KUKA KRL program: MyProgram_006().src

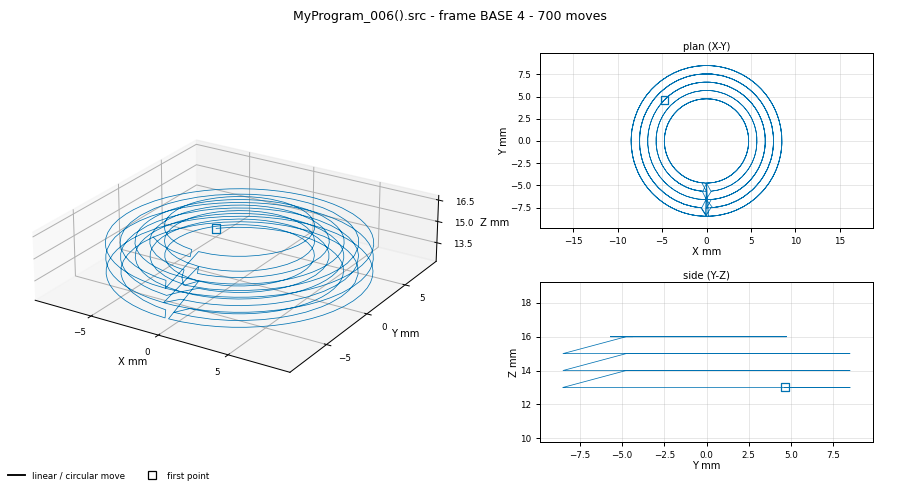
[picture p0: tool path of MyProgram_006().src in frame BASE 4, 700 of 700 moves have a stored position in this frame; points joined in program order, loops and branches not executed]
&ACCESS RVP
&REL 1
&PARAM TEMPLATE = C:\KRC\Roboter\Template\vorgabe
&PARAM EDITMASK = *
DEF MyProgram_006()
; ---- Setting reference (Base) ----
$BASE = BASE_DATA[4]

; --------------------------
; ---- Setting tool (TCP) ----
$TOOL = TOOL_DATA[3]
; --------------------------

$VEL.CP = VEL_APROX_PRINT
Startdeposition()
$VEL.CP = VEL_PRINT
LIN {X -4.726,Y 4.6339,Z 13,A -2.7634,B 0,C 0,E1 0.1598,E2 90.0717} C_DIS
LIN {X -4.1988,Y 5.116,Z 13,A -2.7237,B 0,C 0,E1 0.1598,E2 90.0718} C_DIS
LIN {X -3.6242,Y 5.5404,Z 13,A -2.6847,B 0,C 0,E1 0.1598,E2 90.0719} C_DIS
LIN {X -3.0059,Y 5.8983,Z 13,A -2.6468,B 0,C 0,E1 0.1598,E2 90.0719} C_DIS
LIN {X -2.0359,Y 6.3027,Z 13,A -2.5939,B 0,C 0,E1 0.1598,E2 90.072} C_DIS
LIN {X -1.1961,Y 6.5108,Z 13,A -2.5542,B 0,C 0,E1 0.1598,E2 90.0721} C_DIS
LIN {X -0.51,Y 6.6014,Z 13,A -2.5251,B 0,C 0,E1 0.1598,E2 90.0722} C_DIS
LIN {X 0.1819,Y 6.6196,Z 13,A -2.4988,B 0,C 0,E1 0.1598,E2 90.0722} C_DIS
LIN {X 0.8718,Y 6.5629,Z 13,A -2.4757,B 0,C 0,E1 0.1598,E2 90.0722} C_DIS
LIN {X 1.5516,Y 6.4333,Z 13,A -2.4561,B 0,C 0,E1 0.1598,E2 90.0722} C_DIS
LIN {X 2.2156,Y 6.238,Z 13,A -2.4398,B 0,C 0,E1 0.1598,E2 90.0722} C_DIS
LIN {X 2.8549,Y 5.9732,Z 13,A -2.4274,B 0,C 0,E1 0.1598,E2 90.0722} C_DIS
LIN {X 3.4624,Y 5.6414,Z 13,A -2.419,B 0,C 0,E1 0.1598,E2 90.0722} C_DIS
LIN {X 4.032,Y 5.2483,Z 13,A -2.4146,B 0,C 0,E1 0.1598,E2 90.0722} C_DIS
LIN {X 4.5579,Y 4.7985,Z 13,A -2.4143,B 0,C 0,E1 0.1598,E2 90.0722} C_DIS
LIN {X 5.0373,Y 4.2992,Z 13,A -2.4177,B 0,C 0,E1 0.1598,E2 90.0722} C_DIS
LIN {X 5.4551,Y 3.7474,Z 13,A -2.4257,B 0,C 0,E1 0.1598,E2 90.0722} C_DIS
LIN {X 5.8169,Y 3.1574,Z 13,A -2.4373,B 0,C 0,E1 0.1598,E2 90.0722} C_DIS
LIN {X 6.1152,Y 2.533,Z 13,A -2.4528,B 0,C 0,E1 0.1598,E2 90.0721} C_DIS
LIN {X 6.3464,Y 1.8807,Z 13,A -2.4719,B 0,C 0,E1 0.1598,E2 90.0721} C_DIS
LIN {X 6.5097,Y 1.2082,Z 13,A -2.4944,B 0,C 0,E1 0.1598,E2 90.072} C_DIS
LIN {X 6.6004,Y 0.522,Z 13,A -2.5202,B 0,C 0,E1 0.1598,E2 90.072} C_DIS
LIN {X 6.616,Y -0.1698,Z 13,A -2.549,B 0,C 0,E1 0.1598,E2 90.072} C_DIS
LIN {X 6.5642,Y -0.8599,Z 13,A -2.5802,B 0,C 0,E1 0.1598,E2 90.0719} C_DIS
LIN {X 6.4382,Y -1.5406,Z 13,A -2.6138,B 0,C 0,E1 0.1598,E2 90.0719} C_DIS
LIN {X 6.2414,Y -2.2041,Z 13,A -2.6492,B 0,C 0,E1 0.1598,E2 90.0719} C_DIS
LIN {X 5.9762,Y -2.8433,Z 13,A -2.6861,B 0,C 0,E1 0.1598,E2 90.0718} C_DIS
LIN {X 5.6469,Y -3.4519,Z 13,A -2.7241,B 0,C 0,E1 0.1598,E2 90.0718} C_DIS
LIN {X 5.2569,Y -4.0237,Z 13,A -2.7627,B 0,C 0,E1 0.1598,E2 90.0718} C_DIS
LIN {X 4.8078,Y -4.5503,Z 13,A -2.8016,B 0,C 0,E1 0.1598,E2 90.0717} C_DIS
LIN {X 4.306,Y -5.027,Z 13,A -2.8402,B 0,C 0,E1 0.1598,E2 90.0717} C_DIS
LIN {X 3.7581,Y -5.4501,Z 13,A -2.8783,B 0,C 0,E1 0.1598,E2 90.0717} C_DIS
LIN {X 3.1697,Y -5.8144,Z 13,A -2.9154,B 0,C 0,E1 0.1598,E2 90.0717} C_DIS
LIN {X 2.5442,Y -6.1108,Z 13,A -2.951,B 0,C 0,E1 0.1598,E2 90.0717} C_DIS
LIN {X 1.8922,Y -6.3429,Z 13,A -2.9847,B 0,C 0,E1 0.1598,E2 90.0716} C_DIS
LIN {X 1.2201,Y -6.5075,Z 13,A -3.0164,B 0,C 0,E1 0.1598,E2 90.0716} C_DIS
LIN {X 0.534,Y -6.5994,Z 13,A -3.0455,B 0,C 0,E1 0.1598,E2 90.0716} C_DIS
LIN {X 0.534,Y -6.5994,Z 13,A -3.0455,B 0,C 0,E1 0.1598,E2 90.0716} C_DIS
Enddeposition()
LIN {X -0.0006,Y -7.5571,Z 13,A -3.1047,B 0,C 0,E1 0.1598,E2 90.0703} C_DIS
Startdeposition()
$VEL.CP = VEL_PRINT
LIN {X 1.298,Y -7.4413,Z 13,A -3.0532,B 0,C 0,E1 0.1598,E2 90.0714} C_DIS
LIN {X 2.4367,Y -7.155,Z 13,A -2.9994,B 0,C 0,E1 0.1598,E2 90.0715} C_DIS
LIN {X 3.4286,Y -6.73,Z 13,A -2.9449,B 0,C 0,E1 0.1598,E2 90.0715} C_DIS
LIN {X 4.1743,Y -6.2951,Z 13,A -2.8991,B 0,C 0,E1 0.1598,E2 90.0716} C_DIS
LIN {X 5.1287,Y -5.5503,Z 13,A -2.8322,B 0,C 0,E1 0.1598,E2 90.0716} C_DIS
LIN {X 5.8281,Y -4.8045,Z 13,A -2.7749,B 0,C 0,E1 0.1598,E2 90.0716} C_DIS
LIN {X 6.3134,Y -4.1461,Z 13,A -2.7291,B 0,C 0,E1 0.1598,E2 90.0717} C_DIS
LIN {X 6.8186,Y -3.2572,Z 13,A -2.6725,B 0,C 0,E1 0.1598,E2 90.0715} C_DIS
LIN {X 7.2497,Y -2.1202,Z 13,A -2.6081,B 0,C 0,E1 0.1598,E2 90.0713} C_DIS
LIN {X 7.4278,Y -1.3989,Z 13,A -2.5712,B 0,C 0,E1 0.1598,E2 90.0717} C_DIS
LIN {X 7.5547,Y -0.1838,Z 13,A -2.5146,B 0,C 0,E1 0.1598,E2 90.0715} C_DIS
LIN {X 7.5053,Y 0.8524,Z 13,A -2.4726,B 0,C 0,E1 0.1598,E2 90.0717} C_DIS
LIN {X 7.2814,Y 2.0249,Z 13,A -2.4308,B 0,C 0,E1 0.1598,E2 90.0715} C_DIS
LIN {X 6.7989,Y 3.2979,Z 13,A -2.3945,B 0,C 0,E1 0.1598,E2 90.0715} C_DIS
LIN {X 6.1962,Y 4.3184,Z 13,A -2.3736,B 0,C 0,E1 0.1598,E2 90.0718} C_DIS
LIN {X 5.691,Y 4.9668,Z 13,A -2.3651,B 0,C 0,E1 0.1598,E2 90.0721} C_DIS
LIN {X 5.1177,Y 5.5561,Z 13,A -2.3614,B 0,C 0,E1 0.1598,E2 90.0722} C_DIS
LIN {X 4.483,Y 6.0788,Z 13,A -2.3627,B 0,C 0,E1 0.1598,E2 90.0722} C_DIS
LIN {X 3.795,Y 6.5285,Z 13,A -2.3691,B 0,C 0,E1 0.1598,E2 90.0722} C_DIS
LIN {X 3.0632,Y 6.903,Z 13,A -2.3803,B 0,C 0,E1 0.1598,E2 90.0723} C_DIS
LIN {X 2.0055,Y 7.2865,Z 13,A -2.4031,B 0,C 0,E1 0.1598,E2 90.0723} C_DIS
LIN {X 0.4809,Y 7.5416,Z 13,A -2.4487,B 0,C 0,E1 0.1598,E2 90.0723} C_DIS
LIN {X -1.0225,Y 7.4839,Z 13,A -2.5066,B 0,C 0,E1 0.1598,E2 90.0723} C_DIS
LIN {X -2.1388,Y 7.2487,Z 13,A -2.5577,B 0,C 0,E1 0.1598,E2 90.0721} C_DIS
LIN {X -2.9287,Y 6.966,Z 13,A -2.5988,B 0,C 0,E1 0.1598,E2 90.0721} C_DIS
LIN {X -3.9466,Y 6.441,Z 13,A -2.6584,B 0,C 0,E1 0.1598,E2 90.0719} C_DIS
LIN {X -4.888,Y 5.7626,Z 13,A -2.7216,B 0,C 0,E1 0.1598,E2 90.0717} C_DIS
LIN {X -5.7374,Y 4.9147,Z 13,A -2.7885,B 0,C 0,E1 0.1598,E2 90.0715} C_DIS
LIN {X -6.2527,Y 4.2436,Z 13,A -2.8358,B 0,C 0,E1 0.1598,E2 90.0715} C_DIS
LIN {X -6.9697,Y 2.9199,Z 13,A -2.9174,B 0,C 0,E1 0.1598,E2 90.0709} C_DIS
LIN {X -7.266,Y 2.0827,Z 13,A -2.9641,B 0,C 0,E1 0.1598,E2 90.0713} C_DIS
LIN {X -7.4665,Y 1.165,Z 13,A -3.01,B 0,C 0,E1 0.1598,E2 90.0712} C_DIS
LIN {X -7.5556,Y 0.1435,Z 13,A -3.0562,B 0,C 0,E1 0.1598,E2 90.071} C_DIS
LIN {X -7.5097,Y -0.8431,Z 13,A -3.0961,B 0,C 0,E1 0.1598,E2 90.071} C_DIS
LIN {X -7.2973,Y -1.9496,Z 13,A -3.1347,B 0,C 0,E1 0.1598,E2 90.0708} C_DIS
LIN {X -6.9866,Y -2.8802,Z 13,A -3.1627,B 0,C 0,E1 0.1598,E2 90.0708} C_DIS
LIN {X -6.542,Y -3.7855,Z 13,A -3.1846,B 0,C 0,E1 0.1598,E2 90.0709} C_DIS
LIN {X -5.9161,Y -4.6962,Z 13,A -3.2,B 0,C 0,E1 0.1598,E2 90.0709} C_DIS
LIN {X -5.3836,Y -5.2981,Z 13,A -3.2061,B 0,C 0,E1 0.1598,E2 90.0711} C_DIS
LIN {X -4.6352,Y -5.9679,Z 13,A -3.2069,B 0,C 0,E1 0.1598,E2 90.0711} C_DIS
LIN {X -3.7519,Y -6.5605,Z 13,A -3.1996,B 0,C 0,E1 0.1598,E2 90.0711} C_DIS
LIN {X -2.5893,Y -7.0991,Z 13,A -3.1798,B 0,C 0,E1 0.1598,E2 90.0711} C_DIS
LIN {X -1.4459,Y -7.4139,Z 13,A -3.1513,B 0,C 0,E1 0.1598,E2 90.0713} C_DIS
LIN {X -0.623,Y -7.5271,Z 13,A -3.1259,B 0,C 0,E1 0.1598,E2 90.0713} C_DIS
LIN {X -0.623,Y -7.5271,Z 13,A -3.1259,B 0,C 0,E1 0.1598,E2 90.0714} C_DIS
Enddeposition()
LIN {X -0.0249,Y -8.4916,Z 13,A -3.1439,B 0,C 0,E1 0.1598,E2 90.0702} C_DIS
Startdeposition()
$VEL.CP = VEL_PRINT
LIN {X -1.0697,Y -8.4203,Z 13,A -3.1803,B 0,C 0,E1 0.1598,E2 90.0713} C_DIS
LIN {X -1.8946,Y -8.2735,Z 13,A -3.2044,B 0,C 0,E1 0.1598,E2 90.0713} C_DIS
LIN {X -2.701,Y -8.046,Z 13,A -3.2243,B 0,C 0,E1 0.1598,E2 90.0713} C_DIS
LIN {X -3.4812,Y -7.7404,Z 13,A -3.2399,B 0,C 0,E1 0.1598,E2 90.0712} C_DIS
LIN {X -4.2275,Y -7.3595,Z 13,A -3.2511,B 0,C 0,E1 0.1598,E2 90.0712} C_DIS
LIN {X -4.9328,Y -6.9071,Z 13,A -3.2579,B 0,C 0,E1 0.1598,E2 90.0712} C_DIS
LIN {X -5.5902,Y -6.3876,Z 13,A -3.26,B 0,C 0,E1 0.1598,E2 90.0711} C_DIS
LIN {X -6.1932,Y -5.8058,Z 13,A -3.2575,B 0,C 0,E1 0.1598,E2 90.0711} C_DIS
LIN {X -6.7358,Y -5.1673,Z 13,A -3.2504,B 0,C 0,E1 0.1598,E2 90.0711} C_DIS
LIN {X -7.2124,Y -4.4781,Z 13,A -3.2388,B 0,C 0,E1 0.1598,E2 90.0711} C_DIS
LIN {X -7.7109,Y -3.5571,Z 13,A -3.218,B 0,C 0,E1 0.1598,E2 90.0708} C_DIS
LIN {X -8.1234,Y -2.459,Z 13,A -3.1868,B 0,C 0,E1 0.1598,E2 90.0707} C_DIS
LIN {X -8.3166,Y -1.6994,Z 13,A -3.1622,B 0,C 0,E1 0.1598,E2 90.071} C_DIS
LIN {X -8.4605,Y -0.7301,Z 13,A -3.1264,B 0,C 0,E1 0.1598,E2 90.0708} C_DIS
LIN {X -8.4883,Y 0.1974,Z 13,A -3.0886,B 0,C 0,E1 0.1598,E2 90.071} C_DIS
LIN {X -8.3982,Y 1.2515,Z 13,A -3.0407,B 0,C 0,E1 0.1598,E2 90.071} C_DIS
LIN {X -8.0648,Y 2.6569,Z 13,A -2.9689,B 0,C 0,E1 0.1598,E2 90.0706} C_DIS
LIN {X -7.6043,Y 3.7708,Z 13,A -2.9053,B 0,C 0,E1 0.1598,E2 90.071} C_DIS
LIN {X -7.187,Y 4.5169,Z 13,A -2.8589,B 0,C 0,E1 0.1598,E2 90.0715} C_DIS
LIN {X -6.6963,Y 5.2169,Z 13,A -2.8114,B 0,C 0,E1 0.1598,E2 90.0715} C_DIS
LIN {X -6.1379,Y 5.8643,Z 13,A -2.7636,B 0,C 0,E1 0.1598,E2 90.0717} C_DIS
LIN {X -5.3548,Y 6.5912,Z 13,A -2.704,B 0,C 0,E1 0.1598,E2 90.0717} C_DIS
LIN {X -4.3943,Y 7.2612,Z 13,A -2.6405,B 0,C 0,E1 0.1598,E2 90.0718} C_DIS
LIN {X -3.6905,Y 7.6442,Z 13,A -2.5985,B 0,C 0,E1 0.1598,E2 90.072} C_DIS
LIN {X -2.9534,Y 7.9586,Z 13,A -2.558,B 0,C 0,E1 0.1598,E2 90.0721} C_DIS
LIN {X -1.8584,Y 8.2853,Z 13,A -2.5038,B 0,C 0,E1 0.1598,E2 90.0721} C_DIS
LIN {X -0.8722,Y 8.4432,Z 13,A -2.4608,B 0,C 0,E1 0.1598,E2 90.0723} C_DIS
LIN {X -0.0744,Y 8.4877,Z 13,A -2.4294,B 0,C 0,E1 0.1598,E2 90.0723} C_DIS
LIN {X 0.7241,Y 8.4564,Z 13,A -2.4013,B 0,C 0,E1 0.1598,E2 90.0723} C_DIS
LIN {X 1.5161,Y 8.3505,Z 13,A -2.3765,B 0,C 0,E1 0.1598,E2 90.0723} C_DIS
LIN {X 2.4875,Y 8.1178,Z 13,A -2.3504,B 0,C 0,E1 0.1598,E2 90.0723} C_DIS
LIN {X 3.4541,Y 7.7571,Z 13,A -2.3299,B 0,C 0,E1 0.1598,E2 90.0723} C_DIS
LIN {X 4.4059,Y 7.2529,Z 13,A -2.3161,B 0,C 0,E1 0.1598,E2 90.0723} C_DIS
LIN {X 5.118,Y 6.768,Z 13,A -2.3103,B 0,C 0,E1 0.1598,E2 90.0723} C_DIS
LIN {X 5.7785,Y 6.2148,Z 13,A -2.3093,B 0,C 0,E1 0.1598,E2 90.0723} C_DIS
LIN {X 6.3795,Y 5.5973,Z 13,A -2.3133,B 0,C 0,E1 0.1598,E2 90.0723} C_DIS
LIN {X 6.9145,Y 4.922,Z 13,A -2.3221,B 0,C 0,E1 0.1598,E2 90.0722} C_DIS
LIN {X 7.378,Y 4.1956,Z 13,A -2.3358,B 0,C 0,E1 0.1598,E2 90.0722} C_DIS
LIN {X 7.7655,Y 3.426,Z 13,A -2.3542,B 0,C 0,E1 0.1598,E2 90.0721} C_DIS
LIN {X 8.0732,Y 2.6211,Z 13,A -2.377,B 0,C 0,E1 0.1598,E2 90.0721} C_DIS
LIN {X 8.298,Y 1.7891,Z 13,A -2.404,B 0,C 0,E1 0.1598,E2 90.072} C_DIS
LIN {X 8.461,Y 0.7244,Z 13,A -2.4429,B 0,C 0,E1 0.1598,E2 90.0716} C_DIS
LIN {X 8.4856,Y -0.3159,Z 13,A -2.4863,B 0,C 0,E1 0.1598,E2 90.0716} C_DIS
LIN {X 8.3973,Y -1.2573,Z 13,A -2.5296,B 0,C 0,E1 0.1598,E2 90.0716} C_DIS
LIN {X 8.1747,Y -2.284,Z 13,A -2.5815,B 0,C 0,E1 0.1598,E2 90.0716} C_DIS
LIN {X 7.9086,Y -3.0813,Z 13,A -2.6253,B 0,C 0,E1 0.1598,E2 90.0717} C_DIS
LIN {X 7.565,Y -3.8484,Z 13,A -2.6706,B 0,C 0,E1 0.1598,E2 90.0717} C_DIS
LIN {X 7.1474,Y -4.5778,Z 13,A -2.717,B 0,C 0,E1 0.1598,E2 90.0717} C_DIS
LIN {X 6.6599,Y -5.2624,Z 13,A -2.764,B 0,C 0,E1 0.1598,E2 90.0717} C_DIS
LIN {X 6.1072,Y -5.8957,Z 13,A -2.8112,B 0,C 0,E1 0.1598,E2 90.0717} C_DIS
LIN {X 5.4946,Y -6.4712,Z 13,A -2.8582,B 0,C 0,E1 0.1598,E2 90.0717} C_DIS
LIN {X 4.8279,Y -6.9829,Z 13,A -2.9044,B 0,C 0,E1 0.1598,E2 90.0716} C_DIS
LIN {X 4.1137,Y -7.4261,Z 13,A -2.9495,B 0,C 0,E1 0.1598,E2 90.0716} C_DIS
LIN {X 3.3592,Y -7.7963,Z 13,A -2.9929,B 0,C 0,E1 0.1598,E2 90.0716} C_DIS
LIN {X 2.3714,Y -8.1541,Z 13,A -3.0443,B 0,C 0,E1 0.1598,E2 90.0715} C_DIS
LIN {X 1.132,Y -8.4113,Z 13,A -3.1007,B 0,C 0,E1 0.1598,E2 90.0715} C_DIS
LIN {X 0.2231,Y -8.4876,Z 13,A -3.1372,B 0,C 0,E1 0.1598,E2 90.0714} C_DIS
LIN {X 0.2231,Y -8.4876,Z 13,A -3.1372,B 0,C 0,E1 0.1598,E2 90.0714} C_DIS
Enddeposition()
LIN {X 0.0003,Y -4.7572,Z 14,A -2.9721,B 0,C 0,E1 0.1598,E2 90.0604} C_DIS
Startdeposition()
$VEL.CP = VEL_PRINT
LIN {X 0.0003,Y -4.7572,Z 14,A -2.9778,B 0,C 0,E1 0.1598,E2 90.0661} C_DIS
LIN {X 0.8631,Y -4.6723,Z 14,A -2.9473,B 0,C 0,E1 0.1598,E2 90.071} C_DIS
LIN {X 1.5345,Y -4.4973,Z 14,A -2.9159,B 0,C 0,E1 0.1598,E2 90.0716} C_DIS
LIN {X 2.1731,Y -4.2263,Z 14,A -2.881,B 0,C 0,E1 0.1598,E2 90.0716} C_DIS
LIN {X 2.7641,Y -3.8629,Z 14,A -2.8438,B 0,C 0,E1 0.1598,E2 90.0717} C_DIS
LIN {X 3.3585,Y -3.3581,Z 14,A -2.8005,B 0,C 0,E1 0.1598,E2 90.0717} C_DIS
LIN {X 3.76,Y -2.903,Z 14,A -2.7665,B 0,C 0,E1 0.1598,E2 90.0717} C_DIS
LIN {X 4.1429,Y -2.3248,Z 14,A -2.7278,B 0,C 0,E1 0.1598,E2 90.0717} C_DIS
LIN {X 4.437,Y -1.6966,Z 14,A -2.6903,B 0,C 0,E1 0.1598,E2 90.0717} C_DIS
LIN {X 4.6377,Y -1.0327,Z 14,A -2.6547,B 0,C 0,E1 0.1598,E2 90.0717} C_DIS
LIN {X 4.7394,Y -0.3464,Z 14,A -2.6218,B 0,C 0,E1 0.1598,E2 90.0718} C_DIS
LIN {X 4.7389,Y 0.3474,Z 14,A -2.5924,B 0,C 0,E1 0.1598,E2 90.0718} C_DIS
LIN {X 4.635,Y 1.0331,Z 14,A -2.5672,B 0,C 0,E1 0.1598,E2 90.0718} C_DIS
LIN {X 4.4364,Y 1.6975,Z 14,A -2.5463,B 0,C 0,E1 0.1598,E2 90.0719} C_DIS
LIN {X 4.1422,Y 2.3253,Z 14,A -2.5306,B 0,C 0,E1 0.1598,E2 90.0719} C_DIS
LIN {X 3.7611,Y 2.9048,Z 14,A -2.5201,B 0,C 0,E1 0.1598,E2 90.072} C_DIS
LIN {X 3.2976,Y 3.421,Z 14,A -2.5153,B 0,C 0,E1 0.1598,E2 90.072} C_DIS
LIN {X 2.764,Y 3.8641,Z 14,A -2.5163,B 0,C 0,E1 0.1598,E2 90.072} C_DIS
LIN {X 2.1719,Y 4.2257,Z 14,A -2.5228,B 0,C 0,E1 0.1598,E2 90.0721} C_DIS
LIN {X 1.533,Y 4.4955,Z 14,A -2.535,B 0,C 0,E1 0.1598,E2 90.0721} C_DIS
LIN {X 0.8621,Y 4.6708,Z 14,A -2.5524,B 0,C 0,E1 0.1598,E2 90.0721} C_DIS
LIN {X -0.0007,Y 4.75,Z 14,A -2.5808,B 0,C 0,E1 0.1598,E2 90.0721} C_DIS
LIN {X -0.8635,Y 4.6721,Z 14,A -2.6159,B 0,C 0,E1 0.1598,E2 90.0721} C_DIS
LIN {X -1.5347,Y 4.4969,Z 14,A -2.6481,B 0,C 0,E1 0.1598,E2 90.0721} C_DIS
LIN {X -2.1728,Y 4.2251,Z 14,A -2.683,B 0,C 0,E1 0.1598,E2 90.072} C_DIS
LIN {X -2.7657,Y 3.865,Z 14,A -2.7201,B 0,C 0,E1 0.1598,E2 90.0719} C_DIS
LIN {X -3.2967,Y 3.4188,Z 14,A -2.7584,B 0,C 0,E1 0.1598,E2 90.0718} C_DIS
LIN {X -3.7598,Y 2.9027,Z 14,A -2.7972,B 0,C 0,E1 0.1598,E2 90.0718} C_DIS
LIN {X -4.1837,Y 2.2481,Z 14,A -2.8403,B 0,C 0,E1 0.1598,E2 90.0716} C_DIS
LIN {X -4.4382,Y 1.697,Z 14,A -2.873,B 0,C 0,E1 0.1598,E2 90.0716} C_DIS
LIN {X -4.6371,Y 1.0324,Z 14,A -2.9083,B 0,C 0,E1 0.1598,E2 90.0715} C_DIS
LIN {X -4.7426,Y 0.2596,Z 14,A -2.9447,B 0,C 0,E1 0.1598,E2 90.0713} C_DIS
LIN {X -4.7381,Y -0.3473,Z 14,A -2.9702,B 0,C 0,E1 0.1598,E2 90.0713} C_DIS
LIN {X -4.6366,Y -1.0333,Z 14,A -2.9954,B 0,C 0,E1 0.1598,E2 90.0713} C_DIS
LIN {X -4.4356,Y -1.6968,Z 14,A -3.0161,B 0,C 0,E1 0.1598,E2 90.0713} C_DIS
LIN {X -4.143,Y -2.3255,Z 14,A -3.0319,B 0,C 0,E1 0.1598,E2 90.0713} C_DIS
LIN {X -3.7613,Y -2.9047,Z 14,A -3.0423,B 0,C 0,E1 0.1598,E2 90.0713} C_DIS
LIN {X -3.2979,Y -3.421,Z 14,A -3.0472,B 0,C 0,E1 0.1598,E2 90.0713} C_DIS
LIN {X -2.7644,Y -3.8644,Z 14,A -3.0463,B 0,C 0,E1 0.1598,E2 90.0714} C_DIS
LIN {X -2.1715,Y -4.2243,Z 14,A -3.0398,B 0,C 0,E1 0.1598,E2 90.0714} C_DIS
LIN {X -1.5333,Y -4.4953,Z 14,A -3.0279,B 0,C 0,E1 0.1598,E2 90.0714} C_DIS
LIN {X -0.8622,Y -4.6704,Z 14,A -3.0107,B 0,C 0,E1 0.1598,E2 90.0715} C_DIS
LIN {X 0.0003,Y -4.7572,Z 14,A -2.9827,B 0,C 0,E1 0.1598,E2 90.0715} C_DIS
Enddeposition()
LIN {X 0.0003,Y -4.7572,Z 14,A -2.9827,B 0,C 0,E1 0.1598,E2 90.0715} C_DIS
Startdeposition()
$VEL.CP = VEL_PRINT
LIN {X -0.4069,Y -5.6752,Z 14,A -3.0361,B 0,C 0,E1 0.1598,E2 90.071} C_DIS
LIN {X -1.4862,Y -5.4871,Z 14,A -3.0682,B 0,C 0,E1 0.1598,E2 90.0714} C_DIS
LIN {X -2.1999,Y -5.2405,Z 14,A -3.084,B 0,C 0,E1 0.1598,E2 90.0714} C_DIS
LIN {X -3.1535,Y -4.7363,Z 14,A -3.0976,B 0,C 0,E1 0.1598,E2 90.0713} C_DIS
LIN {X -3.9693,Y -4.0706,Z 14,A -3.0993,B 0,C 0,E1 0.1598,E2 90.0713} C_DIS
LIN {X -4.5265,Y -3.4387,Z 14,A -3.0931,B 0,C 0,E1 0.1598,E2 90.0713} C_DIS
LIN {X -4.9851,Y -2.7321,Z 14,A -3.0801,B 0,C 0,E1 0.1598,E2 90.0712} C_DIS
LIN {X -5.3346,Y -1.9656,Z 14,A -3.0605,B 0,C 0,E1 0.1598,E2 90.0712} C_DIS
LIN {X -5.5663,Y -1.1556,Z 14,A -3.0348,B 0,C 0,E1 0.1598,E2 90.0712} C_DIS
LIN {X -5.6762,Y -0.3204,Z 14,A -3.0036,B 0,C 0,E1 0.1598,E2 90.0712} C_DIS
LIN {X -5.6613,Y 0.522,Z 14,A -2.9675,B 0,C 0,E1 0.1598,E2 90.0712} C_DIS
LIN {X -5.521,Y 1.3526,Z 14,A -2.9274,B 0,C 0,E1 0.1598,E2 90.0713} C_DIS
LIN {X -5.2594,Y 2.153,Z 14,A -2.884,B 0,C 0,E1 0.1598,E2 90.0714} C_DIS
LIN {X -4.8851,Y 2.9075,Z 14,A -2.8385,B 0,C 0,E1 0.1598,E2 90.0715} C_DIS
LIN {X -4.4014,Y 3.5973,Z 14,A -2.7916,B 0,C 0,E1 0.1598,E2 90.0716} C_DIS
LIN {X -3.9787,Y 4.0674,Z 14,A -2.7563,B 0,C 0,E1 0.1598,E2 90.0718} C_DIS
LIN {X -3.0565,Y 4.7945,Z 14,A -2.6915,B 0,C 0,E1 0.1598,E2 90.0718} C_DIS
LIN {X -2.2942,Y 5.2021,Z 14,A -2.6464,B 0,C 0,E1 0.1598,E2 90.072} C_DIS
LIN {X -1.479,Y 5.4897,Z 14,A -2.6042,B 0,C 0,E1 0.1598,E2 90.072} C_DIS
LIN {X -0.6298,Y 5.6507,Z 14,A -2.5661,B 0,C 0,E1 0.1598,E2 90.0721} C_DIS
LIN {X 0.1774,Y 5.6872,Z 14,A -2.5348,B 0,C 0,E1 0.1598,E2 90.0721} C_DIS
LIN {X 0.8669,Y 5.6179,Z 14,A -2.5123,B 0,C 0,E1 0.1598,E2 90.0722} C_DIS
LIN {X 1.5965,Y 5.4619,Z 14,A -2.492,B 0,C 0,E1 0.1598,E2 90.0722} C_DIS
LIN {X 2.1826,Y 5.2486,Z 14,A -2.4794,B 0,C 0,E1 0.1598,E2 90.0722} C_DIS
LIN {X 2.9239,Y 4.8734,Z 14,A -2.4679,B 0,C 0,E1 0.1598,E2 90.0722} C_DIS
LIN {X 3.6041,Y 4.3964,Z 14,A -2.4629,B 0,C 0,E1 0.1598,E2 90.0722} C_DIS
LIN {X 4.2068,Y 3.8244,Z 14,A -2.4649,B 0,C 0,E1 0.1598,E2 90.0721} C_DIS
LIN {X 4.7192,Y 3.1703,Z 14,A -2.4736,B 0,C 0,E1 0.1598,E2 90.0721} C_DIS
LIN {X 5.1305,Y 2.4482,Z 14,A -2.489,B 0,C 0,E1 0.1598,E2 90.072} C_DIS
LIN {X 5.432,Y 1.6742,Z 14,A -2.5107,B 0,C 0,E1 0.1598,E2 90.0719} C_DIS
LIN {X 5.6188,Y 0.8645,Z 14,A -2.5382,B 0,C 0,E1 0.1598,E2 90.0719} C_DIS
LIN {X 5.6873,Y -0.1719,Z 14,A -2.5793,B 0,C 0,E1 0.1598,E2 90.0715} C_DIS
LIN {X 5.5601,Y -1.1791,Z 14,A -2.6269,B 0,C 0,E1 0.1598,E2 90.0715} C_DIS
LIN {X 5.3829,Y -1.8292,Z 14,A -2.6613,B 0,C 0,E1 0.1598,E2 90.0718} C_DIS
LIN {X 5.1291,Y -2.4537,Z 14,A -2.6971,B 0,C 0,E1 0.1598,E2 90.0718} C_DIS
LIN {X 4.7134,Y -3.1865,Z 14,A -2.7434,B 0,C 0,E1 0.1598,E2 90.0716} C_DIS
LIN {X 3.9979,Y -4.0417,Z 14,A -2.8059,B 0,C 0,E1 0.1598,E2 90.0715} C_DIS
LIN {X 3.4096,Y -4.5482,Z 14,A -2.8493,B 0,C 0,E1 0.1598,E2 90.0716} C_DIS
LIN {X 2.7585,Y -4.971,Z 14,A -2.8911,B 0,C 0,E1 0.1598,E2 90.0716} C_DIS
LIN {X 2.0548,Y -5.2988,Z 14,A -2.9309,B 0,C 0,E1 0.1598,E2 90.0716} C_DIS
LIN {X 1.3134,Y -5.5288,Z 14,A -2.9679,B 0,C 0,E1 0.1598,E2 90.0716} C_DIS
LIN {X 0.5478,Y -5.6566,Z 14,A -3.0014,B 0,C 0,E1 0.1598,E2 90.0716} C_DIS
LIN {X 0.5478,Y -5.6566,Z 14,A -3.0014,B 0,C 0,E1 0.1598,E2 90.0716} C_DIS
Enddeposition()
LIN {X -0.0687,Y -6.6224,Z 14,A -3.064,B 0,C 0,E1 0.1598,E2 90.0703} C_DIS
Startdeposition()
$VEL.CP = VEL_PRINT
LIN {X 0.811,Y -6.5699,Z 14,A -3.0306,B 0,C 0,E1 0.1598,E2 90.0715} C_DIS
LIN {X 1.5051,Y -6.4466,Z 14,A -2.9999,B 0,C 0,E1 0.1598,E2 90.0715} C_DIS
LIN {X 2.182,Y -6.2492,Z 14,A -2.9667,B 0,C 0,E1 0.1598,E2 90.0716} C_DIS
LIN {X 2.8348,Y -5.9826,Z 14,A -2.9314,B 0,C 0,E1 0.1598,E2 90.0716} C_DIS
LIN {X 3.4558,Y -5.6487,Z 14,A -2.8945,B 0,C 0,E1 0.1598,E2 90.0716} C_DIS
LIN {X 4.0348,Y -5.2461,Z 14,A -2.8561,B 0,C 0,E1 0.1598,E2 90.0716} C_DIS
LIN {X 4.5708,Y -4.788,Z 14,A -2.8169,B 0,C 0,E1 0.1598,E2 90.0717} C_DIS
LIN {X 5.0545,Y -4.2749,Z 14,A -2.7774,B 0,C 0,E1 0.1598,E2 90.0717} C_DIS
LIN {X 5.4806,Y -3.7132,Z 14,A -2.7378,B 0,C 0,E1 0.1598,E2 90.0717} C_DIS
LIN {X 5.8435,Y -3.1085,Z 14,A -2.6988,B 0,C 0,E1 0.1598,E2 90.0717} C_DIS
LIN {X 6.1397,Y -2.4687,Z 14,A -2.6607,B 0,C 0,E1 0.1598,E2 90.0718} C_DIS
LIN {X 6.3695,Y -1.8022,Z 14,A -2.6239,B 0,C 0,E1 0.1598,E2 90.0718} C_DIS
LIN {X 6.5242,Y -1.1143,Z 14,A -2.589,B 0,C 0,E1 0.1598,E2 90.0718} C_DIS
LIN {X 6.6077,Y -0.4142,Z 14,A -2.5562,B 0,C 0,E1 0.1598,E2 90.0718} C_DIS
LIN {X 6.6125,Y 0.291,Z 14,A -2.526,B 0,C 0,E1 0.1598,E2 90.0719} C_DIS
LIN {X 6.5458,Y 0.9929,Z 14,A -2.4987,B 0,C 0,E1 0.1598,E2 90.0719} C_DIS
LIN {X 6.4037,Y 1.6835,Z 14,A -2.4746,B 0,C 0,E1 0.1598,E2 90.072} C_DIS
LIN {X 6.1878,Y 2.3549,Z 14,A -2.4541,B 0,C 0,E1 0.1598,E2 90.072} C_DIS
LIN {X 5.9018,Y 2.9995,Z 14,A -2.4373,B 0,C 0,E1 0.1598,E2 90.072} C_DIS
LIN {X 5.549,Y 3.6101,Z 14,A -2.4244,B 0,C 0,E1 0.1598,E2 90.0721} C_DIS
LIN {X 5.1339,Y 4.1801,Z 14,A -2.4156,B 0,C 0,E1 0.1598,E2 90.0721} C_DIS
LIN {X 4.6589,Y 4.701,Z 14,A -2.4111,B 0,C 0,E1 0.1598,E2 90.0721} C_DIS
LIN {X 4.1325,Y 5.1701,Z 14,A -2.4106,B 0,C 0,E1 0.1598,E2 90.0722} C_DIS
LIN {X 3.4115,Y 5.6772,Z 14,A -2.4157,B 0,C 0,E1 0.1598,E2 90.0722} C_DIS
LIN {X 2.4839,Y 6.1365,Z 14,A -2.4305,B 0,C 0,E1 0.1598,E2 90.0722} C_DIS
LIN {X 1.819,Y 6.3647,Z 14,A -2.4455,B 0,C 0,E1 0.1598,E2 90.0722} C_DIS
LIN {X 1.1337,Y 6.5215,Z 14,A -2.4642,B 0,C 0,E1 0.1598,E2 90.0722} C_DIS
LIN {X 0.4359,Y 6.6077,Z 14,A -2.4863,B 0,C 0,E1 0.1598,E2 90.0722} C_DIS
LIN {X -0.2671,Y 6.6149,Z 14,A -2.512,B 0,C 0,E1 0.1598,E2 90.0722} C_DIS
LIN {X -0.9671,Y 6.5502,Z 14,A -2.5405,B 0,C 0,E1 0.1598,E2 90.0722} C_DIS
LIN {X -1.6564,Y 6.4118,Z 14,A -2.5718,B 0,C 0,E1 0.1598,E2 90.0722} C_DIS
LIN {X -2.3258,Y 6.1968,Z 14,A -2.6055,B 0,C 0,E1 0.1598,E2 90.0721} C_DIS
LIN {X -2.9695,Y 5.9143,Z 14,A -2.6412,B 0,C 0,E1 0.1598,E2 90.0721} C_DIS
LIN {X -3.5814,Y 5.5684,Z 14,A -2.6783,B 0,C 0,E1 0.1598,E2 90.0719} C_DIS
LIN {X -4.1508,Y 5.1565,Z 14,A -2.7167,B 0,C 0,E1 0.1598,E2 90.0719} C_DIS
LIN {X -4.6745,Y 4.6873,Z 14,A -2.7557,B 0,C 0,E1 0.1598,E2 90.0718} C_DIS
LIN {X -5.1453,Y 4.1652,Z 14,A -2.795,B 0,C 0,E1 0.1598,E2 90.0718} C_DIS
LIN {X -5.5585,Y 3.5965,Z 14,A -2.8342,B 0,C 0,E1 0.1598,E2 90.0716} C_DIS
LIN {X -5.9087,Y 2.987,Z 14,A -2.8728,B 0,C 0,E1 0.1598,E2 90.0716} C_DIS
LIN {X -6.1914,Y 2.3434,Z 14,A -2.9103,B 0,C 0,E1 0.1598,E2 90.0715} C_DIS
LIN {X -6.4037,Y 1.6733,Z 14,A -2.9463,B 0,C 0,E1 0.1598,E2 90.0715} C_DIS
LIN {X -6.5452,Y 0.9847,Z 14,A -2.9805,B 0,C 0,E1 0.1598,E2 90.0714} C_DIS
LIN {X -6.6142,Y 0.2852,Z 14,A -3.0125,B 0,C 0,E1 0.1598,E2 90.0714} C_DIS
LIN {X -6.6072,Y -0.4179,Z 14,A -3.0419,B 0,C 0,E1 0.1598,E2 90.0713} C_DIS
LIN {X -6.5261,Y -1.1162,Z 14,A -3.0683,B 0,C 0,E1 0.1598,E2 90.0713} C_DIS
LIN {X -6.3701,Y -1.8018,Z 14,A -3.0915,B 0,C 0,E1 0.1598,E2 90.0713} C_DIS
LIN {X -6.142,Y -2.4667,Z 14,A -3.1112,B 0,C 0,E1 0.1598,E2 90.0712} C_DIS
LIN {X -5.8459,Y -3.1043,Z 14,A -3.1272,B 0,C 0,E1 0.1598,E2 90.0712} C_DIS
LIN {X -5.2983,Y -3.9745,Z 14,A -3.1437,B 0,C 0,E1 0.1598,E2 90.071} C_DIS
LIN {X -4.7195,Y -4.6427,Z 14,A -3.1508,B 0,C 0,E1 0.1598,E2 90.0712} C_DIS
LIN {X -4.1973,Y -5.1196,Z 14,A -3.1518,B 0,C 0,E1 0.1598,E2 90.0712} C_DIS
LIN {X -3.6266,Y -5.537,Z 14,A -3.1486,B 0,C 0,E1 0.1598,E2 90.0712} C_DIS
LIN {X -3.0152,Y -5.8922,Z 14,A -3.1412,B 0,C 0,E1 0.1598,E2 90.0713} C_DIS
LIN {X -2.205,Y -6.2457,Z 14,A -3.1264,B 0,C 0,E1 0.1598,E2 90.0713} C_DIS
LIN {X -1.1087,Y -6.527,Z 14,A -3.0981,B 0,C 0,E1 0.1598,E2 90.0713} C_DIS
LIN {X -0.0687,Y -6.6224,Z 14,A -3.0641,B 0,C 0,E1 0.1598,E2 90.0715} C_DIS
Enddeposition()
LIN {X -0.0687,Y -6.6224,Z 14,A -3.0641,B 0,C 0,E1 0.1598,E2 90.0715} C_DIS
Startdeposition()
$VEL.CP = VEL_PRINT
LIN {X -0.5385,Y -7.5378,Z 14,A -3.1197,B 0,C 0,E1 0.1598,E2 90.0709} C_DIS
LIN {X -1.7527,Y -7.3469,Z 14,A -3.1566,B 0,C 0,E1 0.1598,E2 90.0713} C_DIS
LIN {X -2.5268,Y -7.1221,Z 14,A -3.1755,B 0,C 0,E1 0.1598,E2 90.0713} C_DIS
LIN {X -3.4486,Y -6.7205,Z 14,A -3.1923,B 0,C 0,E1 0.1598,E2 90.0713} C_DIS
LIN {X -4.1433,Y -6.3149,Z 14,A -3.2006,B 0,C 0,E1 0.1598,E2 90.0713} C_DIS
LIN {X -4.7909,Y -5.8379,Z 14,A -3.2042,B 0,C 0,E1 0.1598,E2 90.0712} C_DIS
LIN {X -5.3842,Y -5.295,Z 14,A -3.203,B 0,C 0,E1 0.1598,E2 90.0712} C_DIS
LIN {X -5.9173,Y -4.6927,Z 14,A -3.1971,B 0,C 0,E1 0.1598,E2 90.0712} C_DIS
LIN {X -6.4926,Y -3.868,Z 14,A -3.1832,B 0,C 0,E1 0.1598,E2 90.0709} C_DIS
LIN {X -6.9575,Y -2.9487,Z 14,A -3.1614,B 0,C 0,E1 0.1598,E2 90.0709} C_DIS
LIN {X -7.3179,Y -1.875,Z 14,A -3.1293,B 0,C 0,E1 0.1598,E2 90.0709} C_DIS
LIN {X -7.5189,Y -0.7604,Z 14,A -3.0895,B 0,C 0,E1 0.1598,E2 90.0707} C_DIS
LIN {X -7.5254,Y 0.7029,Z 14,A -3.0277,B 0,C 0,E1 0.1598,E2 90.0704} C_DIS
LIN {X -7.3869,Y 1.5936,Z 14,A -2.9858,B 0,C 0,E1 0.1598,E2 90.0712} C_DIS
LIN {X -7.0771,Y 2.6353,Z 14,A -2.9304,B 0,C 0,E1 0.1598,E2 90.0711} C_DIS
LIN {X -6.6835,Y 3.5282,Z 14,A -2.8784,B 0,C 0,E1 0.1598,E2 90.0713} C_DIS
LIN {X -5.8869,Y 4.7403,Z 14,A -2.7978,B 0,C 0,E1 0.1598,E2 90.0712} C_DIS
LIN {X -5.2884,Y 5.3972,Z 14,A -2.7485,B 0,C 0,E1 0.1598,E2 90.0717} C_DIS
LIN {X -4.3736,Y 6.1628,Z 14,A -2.6824,B 0,C 0,E1 0.1598,E2 90.0717} C_DIS
LIN {X -3.3752,Y 6.7614,Z 14,A -2.6205,B 0,C 0,E1 0.1598,E2 90.0719} C_DIS
LIN {X -2.3419,Y 7.1808,Z 14,A -2.5647,B 0,C 0,E1 0.1598,E2 90.0721} C_DIS
LIN {X -1.4919,Y 7.4082,Z 14,A -2.5238,B 0,C 0,E1 0.1598,E2 90.0721} C_DIS
LIN {X -0.4422,Y 7.5442,Z 14,A -2.4793,B 0,C 0,E1 0.1598,E2 90.0723} C_DIS
LIN {X 0.5662,Y 7.5359,Z 14,A -2.4425,B 0,C 0,E1 0.1598,E2 90.0723} C_DIS
LIN {X 1.5713,Y 7.3916,Z 14,A -2.4115,B 0,C 0,E1 0.1598,E2 90.0723} C_DIS
LIN {X 2.6378,Y 7.0798,Z 14,A -2.3852,B 0,C 0,E1 0.1598,E2 90.0723} C_DIS
LIN {X 3.4881,Y 6.7042,Z 14,A -2.3697,B 0,C 0,E1 0.1598,E2 90.0723} C_DIS
LIN {X 4.5495,Y 6.0338,Z 14,A -2.3587,B 0,C 0,E1 0.1598,E2 90.0722} C_DIS
LIN {X 5.2007,Y 5.4797,Z 14,A -2.3583,B 0,C 0,E1 0.1598,E2 90.0722} C_DIS
LIN {X 5.9351,Y 4.6777,Z 14,A -2.365,B 0,C 0,E1 0.1598,E2 90.072} C_DIS
LIN {X 6.5048,Y 3.8477,Z 14,A -2.3791,B 0,C 0,E1 0.1598,E2 90.072} C_DIS
LIN {X 7.1657,Y 2.4042,Z 14,A -2.4152,B 0,C 0,E1 0.1598,E2 90.0711} C_DIS
LIN {X 7.4076,Y 1.4951,Z 14,A -2.4456,B 0,C 0,E1 0.1598,E2 90.0718} C_DIS
LIN {X 7.5537,Y 0.2291,Z 14,A -2.4935,B 0,C 0,E1 0.1598,E2 90.0713} C_DIS
LIN {X 7.497,Y -0.9264,Z 14,A -2.5449,B 0,C 0,E1 0.1598,E2 90.0713} C_DIS
LIN {X 7.2981,Y -1.9606,Z 14,A -2.5962,B 0,C 0,E1 0.1598,E2 90.0714} C_DIS
LIN {X 6.8762,Y -3.1245,Z 14,A -2.6611,B 0,C 0,E1 0.1598,E2 90.0712} C_DIS
LIN {X 6.2809,Y -4.2027,Z 14,A -2.729,B 0,C 0,E1 0.1598,E2 90.0714} C_DIS
LIN {X 5.6314,Y -5.034,Z 14,A -2.7884,B 0,C 0,E1 0.1598,E2 90.0715} C_DIS
LIN {X 5.0343,Y -5.6304,Z 14,A -2.8358,B 0,C 0,E1 0.1598,E2 90.0716} C_DIS
LIN {X 4.1035,Y -6.3471,Z 14,A -2.9003,B 0,C 0,E1 0.1598,E2 90.0715} C_DIS
LIN {X 3.2038,Y -6.8399,Z 14,A -2.9544,B 0,C 0,E1 0.1598,E2 90.0715} C_DIS
LIN {X 2.4428,Y -7.1465,Z 14,A -2.9954,B 0,C 0,E1 0.1598,E2 90.0715} C_DIS
LIN {X 1.653,Y -7.3692,Z 14,A -3.0338,B 0,C 0,E1 0.1598,E2 90.0715} C_DIS
LIN {X 0.4884,Y -7.5411,Z 14,A -3.0838,B 0,C 0,E1 0.1598,E2 90.0715} C_DIS
LIN {X 0.4884,Y -7.5411,Z 14,A -3.0838,B 0,C 0,E1 0.1598,E2 90.0715} C_DIS
Enddeposition()
LIN {X -0.1239,Y -8.4891,Z 14,A -3.1455,B 0,C 0,E1 0.1598,E2 90.0702} C_DIS
Startdeposition()
$VEL.CP = VEL_PRINT
LIN {X 0.5639,Y -8.4718,Z 14,A -3.1206,B 0,C 0,E1 0.1598,E2 90.0714} C_DIS
LIN {X 1.5751,Y -8.3447,Z 14,A -3.0782,B 0,C 0,E1 0.1598,E2 90.0714} C_DIS
LIN {X 2.6802,Y -8.0534,Z 14,A -3.0253,B 0,C 0,E1 0.1598,E2 90.0715} C_DIS
LIN {X 3.4659,Y -7.7476,Z 14,A -2.9835,B 0,C 0,E1 0.1598,E2 90.0715} C_DIS
LIN {X 4.2173,Y -7.3652,Z 14,A -2.9397,B 0,C 0,E1 0.1598,E2 90.0715} C_DIS
LIN {X 4.9276,Y -6.9109,Z 14,A -2.8943,B 0,C 0,E1 0.1598,E2 90.0716} C_DIS
LIN {X 5.5893,Y -6.3883,Z 14,A -2.8478,B 0,C 0,E1 0.1598,E2 90.0716} C_DIS
LIN {X 6.4017,Y -5.5771,Z 14,A -2.7834,B 0,C 0,E1 0.1598,E2 90.0716} C_DIS
LIN {X 7.0261,Y -4.761,Z 14,A -2.7257,B 0,C 0,E1 0.1598,E2 90.0716} C_DIS
LIN {X 7.4546,Y -4.0597,Z 14,A -2.6802,B 0,C 0,E1 0.1598,E2 90.0717} C_DIS
LIN {X 7.8125,Y -3.3197,Z 14,A -2.6356,B 0,C 0,E1 0.1598,E2 90.0717} C_DIS
LIN {X 8.0973,Y -2.5486,Z 14,A -2.5923,B 0,C 0,E1 0.1598,E2 90.0717} C_DIS
LIN {X 8.3491,Y -1.5524,Z 14,A -2.5404,B 0,C 0,E1 0.1598,E2 90.0716} C_DIS
LIN {X 8.4728,Y -0.5483,Z 14,A -2.4932,B 0,C 0,E1 0.1598,E2 90.0717} C_DIS
LIN {X 8.4662,Y 0.6212,Z 14,A -2.4435,B 0,C 0,E1 0.1598,E2 90.0715} C_DIS
LIN {X 8.3639,Y 1.4457,Z 14,A -2.4126,B 0,C 0,E1 0.1598,E2 90.0719} C_DIS
LIN {X 8.1814,Y 2.2561,Z 14,A -2.3849,B 0,C 0,E1 0.1598,E2 90.072} C_DIS
LIN {X 7.9213,Y 3.045,Z 14,A -2.361,B 0,C 0,E1 0.1598,E2 90.072} C_DIS
LIN {X 7.5855,Y 3.8048,Z 14,A -2.3411,B 0,C 0,E1 0.1598,E2 90.0721} C_DIS
LIN {X 7.1771,Y 4.5281,Z 14,A -2.3255,B 0,C 0,E1 0.1598,E2 90.0721} C_DIS
LIN {X 6.7002,Y 5.2081,Z 14,A -2.3143,B 0,C 0,E1 0.1598,E2 90.0722} C_DIS
LIN {X 6.1585,Y 5.8377,Z 14,A -2.3076,B 0,C 0,E1 0.1598,E2 90.0722} C_DIS
LIN {X 5.5575,Y 6.4111,Z 14,A -2.3055,B 0,C 0,E1 0.1598,E2 90.0722} C_DIS
LIN {X 4.9053,Y 6.9253,Z 14,A -2.3078,B 0,C 0,E1 0.1598,E2 90.0723} C_DIS
LIN {X 4.025,Y 7.4757,Z 14,A -2.317,B 0,C 0,E1 0.1598,E2 90.0723} C_DIS
LIN {X 2.9607,Y 7.9563,Z 14,A -2.336,B 0,C 0,E1 0.1598,E2 90.0723} C_DIS
LIN {X 2.1648,Y 8.2086,Z 14,A -2.3548,B 0,C 0,E1 0.1598,E2 90.0723} C_DIS
LIN {X 1.348,Y 8.3814,Z 14,A -2.3777,B 0,C 0,E1 0.1598,E2 90.0723} C_DIS
LIN {X 0.5182,Y 8.4723,Z 14,A -2.4046,B 0,C 0,E1 0.1598,E2 90.0723} C_DIS
LIN {X -0.3165,Y 8.4815,Z 14,A -2.435,B 0,C 0,E1 0.1598,E2 90.0723} C_DIS
LIN {X -1.1481,Y 8.4086,Z 14,A -2.4688,B 0,C 0,E1 0.1598,E2 90.0723} C_DIS
LIN {X -1.9685,Y 8.2548,Z 14,A -2.5056,B 0,C 0,E1 0.1598,E2 90.0723} C_DIS
LIN {X -2.77,Y 8.0213,Z 14,A -2.545,B 0,C 0,E1 0.1598,E2 90.0722} C_DIS
LIN {X -3.5447,Y 7.7104,Z 14,A -2.5867,B 0,C 0,E1 0.1598,E2 90.0721} C_DIS
LIN {X -4.2852,Y 7.3251,Z 14,A -2.6302,B 0,C 0,E1 0.1598,E2 90.072} C_DIS
LIN {X -4.9843,Y 6.8689,Z 14,A -2.6752,B 0,C 0,E1 0.1598,E2 90.072} C_DIS
LIN {X -5.6353,Y 6.3463,Z 14,A -2.7212,B 0,C 0,E1 0.1598,E2 90.0718} C_DIS
LIN {X -6.232,Y 5.7625,Z 14,A -2.7678,B 0,C 0,E1 0.1598,E2 90.0718} C_DIS
LIN {X -6.7686,Y 5.1229,Z 14,A -2.8144,B 0,C 0,E1 0.1598,E2 90.0716} C_DIS
LIN {X -7.2381,Y 4.4326,Z 14,A -2.8608,B 0,C 0,E1 0.1598,E2 90.0716} C_DIS
LIN {X -7.7874,Y 3.3828,Z 14,A -2.9249,B 0,C 0,E1 0.1598,E2 90.0712} C_DIS
LIN {X -8.2188,Y 2.13,Z 14,A -2.9932,B 0,C 0,E1 0.1598,E2 90.0708} C_DIS
LIN {X -8.4182,Y 1.1167,Z 14,A -3.0435,B 0,C 0,E1 0.1598,E2 90.071} C_DIS
LIN {X -8.487,Y 0.0681,Z 14,A -3.0902,B 0,C 0,E1 0.1598,E2 90.071} C_DIS
LIN {X -8.4514,Y -0.7719,Z 14,A -3.1243,B 0,C 0,E1 0.1598,E2 90.071} C_DIS
LIN {X -8.2679,Y -1.9391,Z 14,A -3.1665,B 0,C 0,E1 0.1598,E2 90.0707} C_DIS
LIN {X -7.9889,Y -2.8747,Z 14,A -3.1958,B 0,C 0,E1 0.1598,E2 90.0708} C_DIS
LIN {X -7.5802,Y -3.8173,Z 14,A -3.2206,B 0,C 0,E1 0.1598,E2 90.0708} C_DIS
LIN {X -7.1752,Y -4.5324,Z 14,A -3.236,B 0,C 0,E1 0.1598,E2 90.071} C_DIS
LIN {X -6.7029,Y -5.2049,Z 14,A -3.2471,B 0,C 0,E1 0.1598,E2 90.071} C_DIS
LIN {X -6.1682,Y -5.829,Z 14,A -3.2538,B 0,C 0,E1 0.1598,E2 90.071} C_DIS
LIN {X -5.5759,Y -6.3986,Z 14,A -3.2562,B 0,C 0,E1 0.1598,E2 90.071} C_DIS
LIN {X -4.9311,Y -6.908,Z 14,A -3.2541,B 0,C 0,E1 0.1598,E2 90.071} C_DIS
LIN {X -4.2399,Y -7.3523,Z 14,A -3.2475,B 0,C 0,E1 0.1598,E2 90.0711} C_DIS
LIN {X -3.5089,Y -7.7276,Z 14,A -3.2366,B 0,C 0,E1 0.1598,E2 90.0711} C_DIS
LIN {X -2.7451,Y -8.0307,Z 14,A -3.2215,B 0,C 0,E1 0.1598,E2 90.0712} C_DIS
LIN {X -1.9557,Y -8.2586,Z 14,A -3.2022,B 0,C 0,E1 0.1598,E2 90.0712} C_DIS
LIN {X -1.1479,Y -8.409,Z 14,A -3.179,B 0,C 0,E1 0.1598,E2 90.0713} C_DIS
LIN {X -0.1239,Y -8.4891,Z 14,A -3.1449,B 0,C 0,E1 0.1598,E2 90.0713} C_DIS
Enddeposition()
LIN {X 0.0003,Y -4.7572,Z 15,A -2.967,B 0,C 0,E1 0.1598,E2 90.0604} C_DIS
Startdeposition()
$VEL.CP = VEL_PRINT
LIN {X 0.0003,Y -4.7572,Z 15,A -2.9726,B 0,C 0,E1 0.1598,E2 90.0661} C_DIS
LIN {X -0.9367,Y -4.6567,Z 15,A -3.0076,B 0,C 0,E1 0.1598,E2 90.0709} C_DIS
LIN {X -1.8377,Y -4.3814,Z 15,A -3.0296,B 0,C 0,E1 0.1598,E2 90.0714} C_DIS
LIN {X -2.4487,Y -4.0701,Z 15,A -3.0389,B 0,C 0,E1 0.1598,E2 90.0714} C_DIS
LIN {X -3.0107,Y -3.6774,Z 15,A -3.0429,B 0,C 0,E1 0.1598,E2 90.0714} C_DIS
LIN {X -3.508,Y -3.2051,Z 15,A -3.0412,B 0,C 0,E1 0.1598,E2 90.0714} C_DIS
LIN {X -3.9331,Y -2.6672,Z 15,A -3.034,B 0,C 0,E1 0.1598,E2 90.0714} C_DIS
LIN {X -4.2751,Y -2.0728,Z 15,A -3.0215,B 0,C 0,E1 0.1598,E2 90.0714} C_DIS
LIN {X -4.5301,Y -1.4363,Z 15,A -3.0039,B 0,C 0,E1 0.1598,E2 90.0714} C_DIS
LIN {X -4.6881,Y -0.769,Z 15,A -2.9816,B 0,C 0,E1 0.1598,E2 90.0714} C_DIS
LIN {X -4.7496,Y -0.0863,Z 15,A -2.955,B 0,C 0,E1 0.1598,E2 90.0714} C_DIS
LIN {X -4.7155,Y 0.5985,Z 15,A -2.9249,B 0,C 0,E1 0.1598,E2 90.0714} C_DIS
LIN {X -4.5531,Y 1.3526,Z 15,A -2.887,B 0,C 0,E1 0.1598,E2 90.0714} C_DIS
LIN {X -4.3458,Y 1.9155,Z 15,A -2.8557,B 0,C 0,E1 0.1598,E2 90.0716} C_DIS
LIN {X -4.0256,Y 2.5217,Z 15,A -2.8184,B 0,C 0,E1 0.1598,E2 90.0716} C_DIS
LIN {X -3.6213,Y 3.0753,Z 15,A -2.7801,B 0,C 0,E1 0.1598,E2 90.0717} C_DIS
LIN {X -3.1415,Y 3.5653,Z 15,A -2.7418,B 0,C 0,E1 0.1598,E2 90.0717} C_DIS
LIN {X -2.5952,Y 3.9793,Z 15,A -2.7043,B 0,C 0,E1 0.1598,E2 90.0719} C_DIS
LIN {X -1.9958,Y 4.3125,Z 15,A -2.6681,B 0,C 0,E1 0.1598,E2 90.0719} C_DIS
LIN {X -1.1885,Y 4.5985,Z 15,A -2.6263,B 0,C 0,E1 0.1598,E2 90.072} C_DIS
LIN {X -0.5142,Y 4.7214,Z 15,A -2.5963,B 0,C 0,E1 0.1598,E2 90.0721} C_DIS
LIN {X -0.0007,Y 4.7522,Z 15,A -2.5761,B 0,C 0,E1 0.1598,E2 90.0721} C_DIS
LIN {X 0.6831,Y 4.7017,Z 15,A -2.553,B 0,C 0,E1 0.1598,E2 90.0721} C_DIS
LIN {X 1.3528,Y 4.5544,Z 15,A -2.5345,B 0,C 0,E1 0.1598,E2 90.0721} C_DIS
LIN {X 1.9946,Y 4.3129,Z 15,A -2.521,B 0,C 0,E1 0.1598,E2 90.0721} C_DIS
LIN {X 2.5935,Y 3.9789,Z 15,A -2.5131,B 0,C 0,E1 0.1598,E2 90.0721} C_DIS
LIN {X 3.2033,Y 3.5072,Z 15,A -2.5105,B 0,C 0,E1 0.1598,E2 90.0721} C_DIS
LIN {X 3.6202,Y 3.0757,Z 15,A -2.5134,B 0,C 0,E1 0.1598,E2 90.0721} C_DIS
LIN {X 4.0697,Y 2.4495,Z 15,A -2.5233,B 0,C 0,E1 0.1598,E2 90.072} C_DIS
LIN {X 4.348,Y 1.9178,Z 15,A -2.5356,B 0,C 0,E1 0.1598,E2 90.072} C_DIS
LIN {X 4.5763,Y 1.2713,Z 15,A -2.5546,B 0,C 0,E1 0.1598,E2 90.072} C_DIS
LIN {X 4.7115,Y 0.5992,Z 15,A -2.5781,B 0,C 0,E1 0.1598,E2 90.0719} C_DIS
LIN {X 4.7488,Y -0.0852,Z 15,A -2.6057,B 0,C 0,E1 0.1598,E2 90.0719} C_DIS
LIN {X 4.6883,Y -0.768,Z 15,A -2.6369,B 0,C 0,E1 0.1598,E2 90.0719} C_DIS
LIN {X 4.4734,Y -1.5971,Z 15,A -2.6799,B 0,C 0,E1 0.1598,E2 90.0716} C_DIS
LIN {X 4.1136,Y -2.3745,Z 15,A -2.7261,B 0,C 0,E1 0.1598,E2 90.0716} C_DIS
LIN {X 3.7297,Y -2.9425,Z 15,A -2.7645,B 0,C 0,E1 0.1598,E2 90.0717} C_DIS
LIN {X 3.204,Y -3.5065,Z 15,A -2.8077,B 0,C 0,E1 0.1598,E2 90.0717} C_DIS
LIN {X 2.6657,Y -3.9311,Z 15,A -2.8456,B 0,C 0,E1 0.1598,E2 90.0717} C_DIS
LIN {X 2.1491,Y -4.236,Z 15,A -2.8775,B 0,C 0,E1 0.1598,E2 90.0717} C_DIS
LIN {X 1.5177,Y -4.5037,Z 15,A -2.9121,B 0,C 0,E1 0.1598,E2 90.0717} C_DIS
LIN {X 0.8537,Y -4.6758,Z 15,A -2.9438,B 0,C 0,E1 0.1598,E2 90.0717} C_DIS
LIN {X 0.0003,Y -4.7572,Z 15,A -2.9786,B 0,C 0,E1 0.1598,E2 90.0717} C_DIS
Enddeposition()
LIN {X 0.0003,Y -4.7572,Z 15,A -2.9786,B 0,C 0,E1 0.1598,E2 90.0717} C_DIS
Startdeposition()
$VEL.CP = VEL_PRINT
LIN {X 0.4959,Y -5.6627,Z 15,A -2.9983,B 0,C 0,E1 0.1598,E2 90.071} C_DIS
LIN {X 1.1629,Y -5.5669,Z 15,A -2.9703,B 0,C 0,E1 0.1598,E2 90.0716} C_DIS
LIN {X 1.8123,Y -5.388,Z 15,A -2.9389,B 0,C 0,E1 0.1598,E2 90.0716} C_DIS
LIN {X 2.8315,Y -4.9357,Z 15,A -2.8822,B 0,C 0,E1 0.1598,E2 90.0716} C_DIS
LIN {X 3.5385,Y -4.4481,Z 15,A -2.8356,B 0,C 0,E1 0.1598,E2 90.0716} C_DIS
LIN {X 4.0497,Y -3.9892,Z 15,A -2.7973,B 0,C 0,E1 0.1598,E2 90.0717} C_DIS
LIN {X 4.5013,Y -3.4714,Z 15,A -2.7587,B 0,C 0,E1 0.1598,E2 90.0717} C_DIS
LIN {X 4.8888,Y -2.904,Z 15,A -2.7203,B 0,C 0,E1 0.1598,E2 90.0717} C_DIS
LIN {X 5.2024,Y -2.2926,Z 15,A -2.6828,B 0,C 0,E1 0.1598,E2 90.0717} C_DIS
LIN {X 5.4421,Y -1.6487,Z 15,A -2.6467,B 0,C 0,E1 0.1598,E2 90.0718} C_DIS
LIN {X 5.6323,Y -0.8111,Z 15,A -2.6039,B 0,C 0,E1 0.1598,E2 90.0717} C_DIS
LIN {X 5.6716,Y 0.4042,Z 15,A -2.5505,B 0,C 0,E1 0.1598,E2 90.0714} C_DIS
LIN {X 5.5607,Y 1.1821,Z 15,A -2.522,B 0,C 0,E1 0.1598,E2 90.0718} C_DIS
LIN {X 5.342,Y 1.9366,Z 15,A -2.4981,B 0,C 0,E1 0.1598,E2 90.0719} C_DIS
LIN {X 5.0244,Y 2.6549,Z 15,A -2.4793,B 0,C 0,E1 0.1598,E2 90.0719} C_DIS
LIN {X 4.6106,Y 3.3225,Z 15,A -2.4663,B 0,C 0,E1 0.1598,E2 90.072} C_DIS
LIN {X 4.1085,Y 3.9265,Z 15,A -2.4593,B 0,C 0,E1 0.1598,E2 90.072} C_DIS
LIN {X 3.5283,Y 4.4561,Z 15,A -2.4582,B 0,C 0,E1 0.1598,E2 90.0721} C_DIS
LIN {X 2.8797,Y 4.8992,Z 15,A -2.4635,B 0,C 0,E1 0.1598,E2 90.0721} C_DIS
LIN {X 2.1772,Y 5.251,Z 15,A -2.4745,B 0,C 0,E1 0.1598,E2 90.0721} C_DIS
LIN {X 1.1257,Y 5.5772,Z 15,A -2.4995,B 0,C 0,E1 0.1598,E2 90.0721} C_DIS
LIN {X 0.4686,Y 5.666,Z 15,A -2.5201,B 0,C 0,E1 0.1598,E2 90.0721} C_DIS
LIN {X -0.276,Y 5.684,Z 15,A -2.5468,B 0,C 0,E1 0.1598,E2 90.0721} C_DIS
LIN {X -1.2814,Y 5.537,Z 15,A -2.5901,B 0,C 0,E1 0.1598,E2 90.0721} C_DIS
LIN {X -2.0581,Y 5.297,Z 15,A -2.6288,B 0,C 0,E1 0.1598,E2 90.0721} C_DIS
LIN {X -2.7931,Y 4.9499,Z 15,A -2.6705,B 0,C 0,E1 0.1598,E2 90.072} C_DIS
LIN {X -3.4701,Y 4.5002,Z 15,A -2.7144,B 0,C 0,E1 0.1598,E2 90.0719} C_DIS
LIN {X -4.0769,Y 3.9596,Z 15,A -2.7595,B 0,C 0,E1 0.1598,E2 90.0717} C_DIS
LIN {X -4.6012,Y 3.3382,Z 15,A -2.805,B 0,C 0,E1 0.1598,E2 90.0717} C_DIS
LIN {X -5.0298,Y 2.6475,Z 15,A -2.8499,B 0,C 0,E1 0.1598,E2 90.0715} C_DIS
LIN {X -5.356,Y 1.9029,Z 15,A -2.8932,B 0,C 0,E1 0.1598,E2 90.0715} C_DIS
LIN {X -5.5727,Y 1.1194,Z 15,A -2.9342,B 0,C 0,E1 0.1598,E2 90.0713} C_DIS
LIN {X -5.6749,Y 0.313,Z 15,A -2.9719,B 0,C 0,E1 0.1598,E2 90.0713} C_DIS
LIN {X -5.6602,Y -0.4996,Z 15,A -3.0057,B 0,C 0,E1 0.1598,E2 90.0713} C_DIS
LIN {X -5.5315,Y -1.302,Z 15,A -3.0348,B 0,C 0,E1 0.1598,E2 90.0712} C_DIS
LIN {X -5.2893,Y -2.0779,Z 15,A -3.0586,B 0,C 0,E1 0.1598,E2 90.0712} C_DIS
LIN {X -4.939,Y -2.8114,Z 15,A -3.0768,B 0,C 0,E1 0.1598,E2 90.0712} C_DIS
LIN {X -4.4894,Y -3.4888,Z 15,A -3.0889,B 0,C 0,E1 0.1598,E2 90.0712} C_DIS
LIN {X -3.9456,Y -4.0933,Z 15,A -3.0945,B 0,C 0,E1 0.1598,E2 90.0712} C_DIS
LIN {X -3.1567,Y -4.7341,Z 15,A -3.0926,B 0,C 0,E1 0.1598,E2 90.0712} C_DIS
LIN {X -2.2934,Y -5.2029,Z 15,A -3.0808,B 0,C 0,E1 0.1598,E2 90.0713} C_DIS
LIN {X -1.7072,Y -5.4252,Z 15,A -3.0688,B 0,C 0,E1 0.1598,E2 90.0715} C_DIS
LIN {X -1.0997,Y -5.5793,Z 15,A -3.0531,B 0,C 0,E1 0.1598,E2 90.0715} C_DIS
LIN {X -0.4788,Y -5.6661,Z 15,A -3.034,B 0,C 0,E1 0.1598,E2 90.0715} C_DIS
LIN {X -0.4788,Y -5.6661,Z 15,A -3.034,B 0,C 0,E1 0.1598,E2 90.0715} C_DIS
Enddeposition()
LIN {X -0.009,Y -6.6202,Z 15,A -3.0561,B 0,C 0,E1 0.1598,E2 90.0703} C_DIS
Startdeposition()
$VEL.CP = VEL_PRINT
LIN {X -0.9066,Y -6.5577,Z 15,A -3.0875,B 0,C 0,E1 0.1598,E2 90.0714} C_DIS
LIN {X -1.6134,Y -6.4205,Z 15,A -3.1077,B 0,C 0,E1 0.1598,E2 90.0714} C_DIS
LIN {X -2.3008,Y -6.2065,Z 15,A -3.1238,B 0,C 0,E1 0.1598,E2 90.0714} C_DIS
LIN {X -2.961,Y -5.9195,Z 15,A -3.1359,B 0,C 0,E1 0.1598,E2 90.0714} C_DIS
LIN {X -3.5862,Y -5.5627,Z 15,A -3.1437,B 0,C 0,E1 0.1598,E2 90.0714} C_DIS
LIN {X -4.1693,Y -5.141,Z 15,A -3.1473,B 0,C 0,E1 0.1598,E2 90.0713} C_DIS
LIN {X -4.7029,Y -4.6577,Z 15,A -3.1464,B 0,C 0,E1 0.1598,E2 90.0713} C_DIS
LIN {X -5.2945,Y -3.9795,Z 15,A -3.1393,B 0,C 0,E1 0.1598,E2 90.0711} C_DIS
LIN {X -5.8444,Y -3.1071,Z 15,A -3.1226,B 0,C 0,E1 0.1598,E2 90.071} C_DIS
LIN {X -6.1408,Y -2.4698,Z 15,A -3.1067,B 0,C 0,E1 0.1598,E2 90.0712} C_DIS
LIN {X -6.3692,Y -1.805,Z 15,A -3.0871,B 0,C 0,E1 0.1598,E2 90.0712} C_DIS
LIN {X -6.5254,Y -1.1197,Z 15,A -3.0639,B 0,C 0,E1 0.1598,E2 90.0712} C_DIS
LIN {X -6.6069,Y -0.4215,Z 15,A -3.0375,B 0,C 0,E1 0.1598,E2 90.0712} C_DIS
LIN {X -6.6138,Y 0.2813,Z 15,A -3.0081,B 0,C 0,E1 0.1598,E2 90.0713} C_DIS
LIN {X -6.5478,Y 0.9812,Z 15,A -2.9762,B 0,C 0,E1 0.1598,E2 90.0713} C_DIS
LIN {X -6.4038,Y 1.6691,Z 15,A -2.9419,B 0,C 0,E1 0.1598,E2 90.0714} C_DIS
LIN {X -6.1928,Y 2.3396,Z 15,A -2.9059,B 0,C 0,E1 0.1598,E2 90.0714} C_DIS
LIN {X -5.9107,Y 2.9832,Z 15,A -2.8684,B 0,C 0,E1 0.1598,E2 90.0715} C_DIS
LIN {X -5.5609,Y 3.5928,Z 15,A -2.8298,B 0,C 0,E1 0.1598,E2 90.0716} C_DIS
LIN {X -5.1481,Y 4.1617,Z 15,A -2.7906,B 0,C 0,E1 0.1598,E2 90.0716} C_DIS
LIN {X -4.6776,Y 4.6838,Z 15,A -2.7513,B 0,C 0,E1 0.1598,E2 90.0718} C_DIS
LIN {X -4.1547,Y 5.1535,Z 15,A -2.7123,B 0,C 0,E1 0.1598,E2 90.0718} C_DIS
LIN {X -3.5855,Y 5.5657,Z 15,A -2.6739,B 0,C 0,E1 0.1598,E2 90.0719} C_DIS
LIN {X -2.9741,Y 5.912,Z 15,A -2.6368,B 0,C 0,E1 0.1598,E2 90.072} C_DIS
LIN {X -2.3308,Y 6.1953,Z 15,A -2.6011,B 0,C 0,E1 0.1598,E2 90.072} C_DIS
LIN {X -1.6616,Y 6.4104,Z 15,A -2.5674,B 0,C 0,E1 0.1598,E2 90.0721} C_DIS
LIN {X -0.9726,Y 6.5495,Z 15,A -2.5361,B 0,C 0,E1 0.1598,E2 90.0721} C_DIS
LIN {X -0.2727,Y 6.6145,Z 15,A -2.5075,B 0,C 0,E1 0.1598,E2 90.0722} C_DIS
LIN {X 0.4301,Y 6.6062,Z 15,A -2.4819,B 0,C 0,E1 0.1598,E2 90.0722} C_DIS
LIN {X 1.128,Y 6.5222,Z 15,A -2.4597,B 0,C 0,E1 0.1598,E2 90.0722} C_DIS
LIN {X 1.8133,Y 6.3663,Z 15,A -2.441,B 0,C 0,E1 0.1598,E2 90.0722} C_DIS
LIN {X 2.4783,Y 6.1387,Z 15,A -2.4261,B 0,C 0,E1 0.1598,E2 90.0722} C_DIS
LIN {X 3.4115,Y 5.6772,Z 15,A -2.4111,B 0,C 0,E1 0.1598,E2 90.0722} C_DIS
LIN {X 4.1301,Y 5.172,Z 15,A -2.406,B 0,C 0,E1 0.1598,E2 90.0722} C_DIS
LIN {X 4.6549,Y 4.7048,Z 15,A -2.4064,B 0,C 0,E1 0.1598,E2 90.0722} C_DIS
LIN {X 5.1289,Y 4.1863,Z 15,A -2.4109,B 0,C 0,E1 0.1598,E2 90.0722} C_DIS
LIN {X 5.543,Y 3.6185,Z 15,A -2.4197,B 0,C 0,E1 0.1598,E2 90.0722} C_DIS
LIN {X 5.8958,Y 3.0108,Z 15,A -2.4324,B 0,C 0,E1 0.1598,E2 90.0722} C_DIS
LIN {X 6.1824,Y 2.3691,Z 15,A -2.4491,B 0,C 0,E1 0.1598,E2 90.0721} C_DIS
LIN {X 6.399,Y 1.7005,Z 15,A -2.4694,B 0,C 0,E1 0.1598,E2 90.0721} C_DIS
LIN {X 6.5427,Y 1.0127,Z 15,A -2.4933,B 0,C 0,E1 0.1598,E2 90.072} C_DIS
LIN {X 6.6127,Y 0.3134,Z 15,A -2.5204,B 0,C 0,E1 0.1598,E2 90.072} C_DIS
LIN {X 6.6075,Y -0.3892,Z 15,A -2.5505,B 0,C 0,E1 0.1598,E2 90.0719} C_DIS
LIN {X 6.5292,Y -1.0875,Z 15,A -2.583,B 0,C 0,E1 0.1598,E2 90.0719} C_DIS
LIN {X 6.3779,Y -1.7737,Z 15,A -2.6177,B 0,C 0,E1 0.1598,E2 90.0719} C_DIS
LIN {X 6.1534,Y -2.4396,Z 15,A -2.6543,B 0,C 0,E1 0.1598,E2 90.0718} C_DIS
LIN {X 5.8608,Y -3.0784,Z 15,A -2.6922,B 0,C 0,E1 0.1598,E2 90.0718} C_DIS
LIN {X 5.5022,Y -3.6826,Z 15,A -2.731,B 0,C 0,E1 0.1598,E2 90.0718} C_DIS
LIN {X 5.0806,Y -4.2448,Z 15,A -2.7704,B 0,C 0,E1 0.1598,E2 90.0718} C_DIS
LIN {X 4.6012,Y -4.7585,Z 15,A -2.8099,B 0,C 0,E1 0.1598,E2 90.0717} C_DIS
LIN {X 4.0706,Y -5.2193,Z 15,A -2.8489,B 0,C 0,E1 0.1598,E2 90.0717} C_DIS
LIN {X 3.4961,Y -5.624,Z 15,A -2.8872,B 0,C 0,E1 0.1598,E2 90.0717} C_DIS
LIN {X 2.8798,Y -5.9617,Z 15,A -2.9242,B 0,C 0,E1 0.1598,E2 90.0717} C_DIS
LIN {X 2.231,Y -6.2317,Z 15,A -2.9595,B 0,C 0,E1 0.1598,E2 90.0716} C_DIS
LIN {X 1.5578,Y -6.4329,Z 15,A -2.9927,B 0,C 0,E1 0.1598,E2 90.0716} C_DIS
LIN {X 0.8674,Y -6.5638,Z 15,A -3.0236,B 0,C 0,E1 0.1598,E2 90.0716} C_DIS
LIN {X -0.009,Y -6.6202,Z 15,A -3.0582,B 0,C 0,E1 0.1598,E2 90.0715} C_DIS
Enddeposition()
LIN {X -0.009,Y -6.6202,Z 15,A -3.0582,B 0,C 0,E1 0.1598,E2 90.0715} C_DIS
Startdeposition()
$VEL.CP = VEL_PRINT
LIN {X 0.6964,Y -7.5205,Z 15,A -3.0701,B 0,C 0,E1 0.1598,E2 90.0709} C_DIS
LIN {X 2.3131,Y -7.1941,Z 15,A -2.9974,B 0,C 0,E1 0.1598,E2 90.0715} C_DIS
LIN {X 3.6078,Y -6.6346,Z 15,A -2.9261,B 0,C 0,E1 0.1598,E2 90.0715} C_DIS
LIN {X 4.2843,Y -6.2184,Z 15,A -2.8837,B 0,C 0,E1 0.1598,E2 90.0716} C_DIS
LIN {X 5.3338,Y -5.3554,Z 15,A -2.8082,B 0,C 0,E1 0.1598,E2 90.0714} C_DIS
LIN {X 6.088,Y -4.4674,Z 15,A -2.7427,B 0,C 0,E1 0.1598,E2 90.0714} C_DIS
LIN {X 6.5371,Y -3.7822,Z 15,A -2.6973,B 0,C 0,E1 0.1598,E2 90.0717} C_DIS
LIN {X 6.9094,Y -3.0522,Z 15,A -2.6526,B 0,C 0,E1 0.1598,E2 90.0717} C_DIS
LIN {X 7.1983,Y -2.2856,Z 15,A -2.6093,B 0,C 0,E1 0.1598,E2 90.0717} C_DIS
LIN {X 7.4052,Y -1.4928,Z 15,A -2.568,B 0,C 0,E1 0.1598,E2 90.0718} C_DIS
LIN {X 7.5419,Y -0.4776,Z 15,A -2.5195,B 0,C 0,E1 0.1598,E2 90.0716} C_DIS
LIN {X 7.5396,Y 0.5112,Z 15,A -2.4777,B 0,C 0,E1 0.1598,E2 90.0717} C_DIS
LIN {X 7.3496,Y 1.7388,Z 15,A -2.4321,B 0,C 0,E1 0.1598,E2 90.0714} C_DIS
LIN {X 6.8571,Y 3.178,Z 15,A -2.3889,B 0,C 0,E1 0.1598,E2 90.0712} C_DIS
LIN {X 6.2053,Y 4.3076,Z 15,A -2.3655,B 0,C 0,E1 0.1598,E2 90.0717} C_DIS
LIN {X 5.5701,Y 5.1078,Z 15,A -2.3552,B 0,C 0,E1 0.1598,E2 90.072} C_DIS
LIN {X 4.7833,Y 5.8522,Z 15,A -2.3528,B 0,C 0,E1 0.1598,E2 90.072} C_DIS
LIN {X 4.0805,Y 6.3613,Z 15,A -2.3573,B 0,C 0,E1 0.1598,E2 90.0722} C_DIS
LIN {X 2.8084,Y 7.0169,Z 15,A -2.3764,B 0,C 0,E1 0.1598,E2 90.0722} C_DIS
LIN {X 1.858,Y 7.3249,Z 15,A -2.3987,B 0,C 0,E1 0.1598,E2 90.0722} C_DIS
LIN {X 0.684,Y 7.5276,Z 15,A -2.4335,B 0,C 0,E1 0.1598,E2 90.0722} C_DIS
LIN {X -0.4985,Y 7.5391,Z 15,A -2.4767,B 0,C 0,E1 0.1598,E2 90.0722} C_DIS
LIN {X -1.2191,Y 7.4543,Z 15,A -2.5069,B 0,C 0,E1 0.1598,E2 90.0722} C_DIS
LIN {X -2.105,Y 7.2593,Z 15,A -2.5478,B 0,C 0,E1 0.1598,E2 90.0722} C_DIS
LIN {X -3.2447,Y 6.8247,Z 15,A -2.6081,B 0,C 0,E1 0.1598,E2 90.072} C_DIS
LIN {X -4.16,Y 6.3032,Z 15,A -2.6638,B 0,C 0,E1 0.1598,E2 90.072} C_DIS
LIN {X -5.2736,Y 5.4127,Z 15,A -2.7421,B 0,C 0,E1 0.1598,E2 90.0715} C_DIS
LIN {X -6.0646,Y 4.5091,Z 15,A -2.8094,B 0,C 0,E1 0.1598,E2 90.0715} C_DIS
LIN {X -6.7097,Y 3.467,Z 15,A -2.8769,B 0,C 0,E1 0.1598,E2 90.0712} C_DIS
LIN {X -7.1166,Y 2.5419,Z 15,A -2.9308,B 0,C 0,E1 0.1598,E2 90.0712} C_DIS
LIN {X -7.4237,Y 1.3908,Z 15,A -2.9904,B 0,C 0,E1 0.1598,E2 90.0708} C_DIS
LIN {X -7.5575,Y -0.0615,Z 15,A -3.0561,B 0,C 0,E1 0.1598,E2 90.0704} C_DIS
LIN {X -7.4267,Y -1.376,Z 15,A -3.1069,B 0,C 0,E1 0.1598,E2 90.0705} C_DIS
LIN {X -7.1578,Y -2.4288,Z 15,A -3.1416,B 0,C 0,E1 0.1598,E2 90.0707} C_DIS
LIN {X -6.7091,Y -3.469,Z 15,A -3.1691,B 0,C 0,E1 0.1598,E2 90.0707} C_DIS
LIN {X -6.1796,Y -4.3492,Z 15,A -3.1869,B 0,C 0,E1 0.1598,E2 90.0708} C_DIS
LIN {X -5.5197,Y -5.161,Z 15,A -3.197,B 0,C 0,E1 0.1598,E2 90.071} C_DIS
LIN {X -4.7565,Y -5.8671,Z 15,A -3.199,B 0,C 0,E1 0.1598,E2 90.071} C_DIS
LIN {X -4.0819,Y -6.3537,Z 15,A -3.1949,B 0,C 0,E1 0.1598,E2 90.0712} C_DIS
LIN {X -3.3585,Y -6.7641,Z 15,A -3.1858,B 0,C 0,E1 0.1598,E2 90.0712} C_DIS
LIN {X -2.4,Y -7.167,Z 15,A -3.1677,B 0,C 0,E1 0.1598,E2 90.0712} C_DIS
LIN {X -1.3364,Y -7.4339,Z 15,A -3.14,B 0,C 0,E1 0.1598,E2 90.0713} C_DIS
LIN {X -0.5681,Y -7.5302,Z 15,A -3.116,B 0,C 0,E1 0.1598,E2 90.0714} C_DIS
LIN {X -0.5681,Y -7.5302,Z 15,A -3.116,B 0,C 0,E1 0.1598,E2 90.0714} C_DIS
Enddeposition()
LIN {X 0.036,Y -8.4913,Z 15,A -3.1336,B 0,C 0,E1 0.1598,E2 90.0702} C_DIS
Startdeposition()
$VEL.CP = VEL_PRINT
LIN {X -0.965,Y -8.4327,Z 15,A -3.1689,B 0,C 0,E1 0.1598,E2 90.0713} C_DIS
LIN {X -1.7571,Y -8.3058,Z 15,A -3.1926,B 0,C 0,E1 0.1598,E2 90.0713} C_DIS
LIN {X -2.5332,Y -8.1023,Z 15,A -3.2124,B 0,C 0,E1 0.1598,E2 90.0713} C_DIS
LIN {X -3.2864,Y -7.8263,Z 15,A -3.2283,B 0,C 0,E1 0.1598,E2 90.0713} C_DIS
LIN {X -4.0104,Y -7.4807,Z 15,A -3.2402,B 0,C 0,E1 0.1598,E2 90.0712} C_DIS
LIN {X -4.6984,Y -7.0684,Z 15,A -3.248,B 0,C 0,E1 0.1598,E2 90.0712} C_DIS
LIN {X -5.3444,Y -6.5929,Z 15,A -3.2516,B 0,C 0,E1 0.1598,E2 90.0712} C_DIS
LIN {X -5.9424,Y -6.0585,Z 15,A -3.2509,B 0,C 0,E1 0.1598,E2 90.0711} C_DIS
LIN {X -6.4875,Y -5.4701,Z 15,A -3.246,B 0,C 0,E1 0.1598,E2 90.0711} C_DIS
LIN {X -6.9751,Y -4.8331,Z 15,A -3.237,B 0,C 0,E1 0.1598,E2 90.0711} C_DIS
LIN {X -7.4007,Y -4.1532,Z 15,A -3.2239,B 0,C 0,E1 0.1598,E2 90.0711} C_DIS
LIN {X -7.7605,Y -3.4362,Z 15,A -3.2069,B 0,C 0,E1 0.1598,E2 90.0711} C_DIS
LIN {X -8.1493,Y -2.387,Z 15,A -3.1767,B 0,C 0,E1 0.1598,E2 90.0708} C_DIS
LIN {X -8.3745,Y -1.3987,Z 15,A -3.1433,B 0,C 0,E1 0.1598,E2 90.0708} C_DIS
LIN {X -8.4797,Y -0.3486,Z 15,A -3.1029,B 0,C 0,E1 0.1598,E2 90.0709} C_DIS
LIN {X -8.4734,Y 0.4955,Z 15,A -3.0673,B 0,C 0,E1 0.1598,E2 90.0711} C_DIS
LIN {X -8.3833,Y 1.335,Z 15,A -3.0287,B 0,C 0,E1 0.1598,E2 90.0711} C_DIS
LIN {X -8.1292,Y 2.4512,Z 15,A -2.9721,B 0,C 0,E1 0.1598,E2 90.0711} C_DIS
LIN {X -7.778,Y 3.4051,Z 15,A -2.9191,B 0,C 0,E1 0.1598,E2 90.0711} C_DIS
LIN {X -7.2942,Y 4.3394,Z 15,A -2.862,B 0,C 0,E1 0.1598,E2 90.0714} C_DIS
LIN {X -6.8279,Y 5.0401,Z 15,A -2.8155,B 0,C 0,E1 0.1598,E2 90.0716} C_DIS
LIN {X -6.2948,Y 5.6914,Z 15,A -2.7684,B 0,C 0,E1 0.1598,E2 90.0716} C_DIS
LIN {X -5.6998,Y 6.2866,Z 15,A -2.7214,B 0,C 0,E1 0.1598,E2 90.0718} C_DIS
LIN {X -5.0489,Y 6.82,Z 15,A -2.675,B 0,C 0,E1 0.1598,E2 90.0718} C_DIS
LIN {X -4.3482,Y 7.2862,Z 15,A -2.6295,B 0,C 0,E1 0.1598,E2 90.072} C_DIS
LIN {X -3.6052,Y 7.6814,Z 15,A -2.5855,B 0,C 0,E1 0.1598,E2 90.072} C_DIS
LIN {X -2.8266,Y 8.0008,Z 15,A -2.5433,B 0,C 0,E1 0.1598,E2 90.0721} C_DIS
LIN {X -2.0202,Y 8.2417,Z 15,A -2.5034,B 0,C 0,E1 0.1598,E2 90.0722} C_DIS
LIN {X -1.1939,Y 8.4016,Z 15,A -2.4661,B 0,C 0,E1 0.1598,E2 90.0722} C_DIS
LIN {X -0.3559,Y 8.4794,Z 15,A -2.4319,B 0,C 0,E1 0.1598,E2 90.0723} C_DIS
LIN {X 0.4857,Y 8.4746,Z 15,A -2.401,B 0,C 0,E1 0.1598,E2 90.0723} C_DIS
LIN {X 1.3228,Y 8.3857,Z 15,A -2.3739,B 0,C 0,E1 0.1598,E2 90.0723} C_DIS
LIN {X 2.1468,Y 8.2136,Z 15,A -2.3507,B 0,C 0,E1 0.1598,E2 90.0724} C_DIS
LIN {X 2.9497,Y 7.9606,Z 15,A -2.3317,B 0,C 0,E1 0.1598,E2 90.0724} C_DIS
LIN {X 4.027,Y 7.4746,Z 15,A -2.3124,B 0,C 0,E1 0.1598,E2 90.0724} C_DIS
LIN {X 4.8972,Y 6.9323,Z 15,A -2.3032,B 0,C 0,E1 0.1598,E2 90.0724} C_DIS
LIN {X 5.5437,Y 6.4272,Z 15,A -2.3008,B 0,C 0,E1 0.1598,E2 90.0724} C_DIS
LIN {X 6.1377,Y 5.8612,Z 15,A -2.3028,B 0,C 0,E1 0.1598,E2 90.0724} C_DIS
LIN {X 6.6751,Y 5.2413,Z 15,A -2.3092,B 0,C 0,E1 0.1598,E2 90.0723} C_DIS
LIN {X 7.1501,Y 4.5723,Z 15,A -2.3201,B 0,C 0,E1 0.1598,E2 90.0723} C_DIS
LIN {X 7.5586,Y 3.8607,Z 15,A -2.3352,B 0,C 0,E1 0.1598,E2 90.0722} C_DIS
LIN {X 7.8961,Y 3.1127,Z 15,A -2.3545,B 0,C 0,E1 0.1598,E2 90.0722} C_DIS
LIN {X 8.1594,Y 2.3356,Z 15,A -2.3777,B 0,C 0,E1 0.1598,E2 90.072} C_DIS
LIN {X 8.3464,Y 1.5367,Z 15,A -2.4048,B 0,C 0,E1 0.1598,E2 90.072} C_DIS
LIN {X 8.4563,Y 0.7237,Z 15,A -2.4353,B 0,C 0,E1 0.1598,E2 90.072} C_DIS
LIN {X 8.4871,Y -0.0961,Z 15,A -2.469,B 0,C 0,E1 0.1598,E2 90.072} C_DIS
LIN {X 8.4398,Y -0.9153,Z 15,A -2.5055,B 0,C 0,E1 0.1598,E2 90.0719} C_DIS
LIN {X 8.3118,Y -1.7258,Z 15,A -2.5447,B 0,C 0,E1 0.1598,E2 90.0719} C_DIS
LIN {X 8.1059,Y -2.52,Z 15,A -2.5861,B 0,C 0,E1 0.1598,E2 90.0718} C_DIS
LIN {X 7.8249,Y -3.2908,Z 15,A -2.6292,B 0,C 0,E1 0.1598,E2 90.0718} C_DIS
LIN {X 7.4699,Y -4.0306,Z 15,A -2.6737,B 0,C 0,E1 0.1598,E2 90.0718} C_DIS
LIN {X 7.0454,Y -4.7326,Z 15,A -2.7192,B 0,C 0,E1 0.1598,E2 90.0717} C_DIS
LIN {X 6.4253,Y -5.5495,Z 15,A -2.7766,B 0,C 0,E1 0.1598,E2 90.0715} C_DIS
LIN {X 5.5869,Y -6.3906,Z 15,A -2.8431,B 0,C 0,E1 0.1598,E2 90.0715} C_DIS
LIN {X 4.931,Y -6.9086,Z 15,A -2.8894,B 0,C 0,E1 0.1598,E2 90.0715} C_DIS
LIN {X 4.2276,Y -7.3599,Z 15,A -2.9344,B 0,C 0,E1 0.1598,E2 90.0715} C_DIS
LIN {X 3.4832,Y -7.74,Z 15,A -2.9779,B 0,C 0,E1 0.1598,E2 90.0715} C_DIS
LIN {X 2.7051,Y -8.045,Z 15,A -3.0194,B 0,C 0,E1 0.1598,E2 90.0715} C_DIS
LIN {X 1.9008,Y -8.2721,Z 15,A -3.0585,B 0,C 0,E1 0.1598,E2 90.0715} C_DIS
LIN {X 1.0781,Y -8.419,Z 15,A -3.0949,B 0,C 0,E1 0.1598,E2 90.0715} C_DIS
LIN {X 0.036,Y -8.4913,Z 15,A -3.1362,B 0,C 0,E1 0.1598,E2 90.0714} C_DIS
Enddeposition()
LIN {X 0.0003,Y -4.7572,Z 16,A -2.964,B 0,C 0,E1 0.1598,E2 90.0603} C_DIS
Startdeposition()
$VEL.CP = VEL_PRINT
LIN {X 0.0003,Y -4.7572,Z 16,A -2.9697,B 0,C 0,E1 0.1598,E2 90.0661} C_DIS
LIN {X 0.8634,Y -4.6735,Z 16,A -2.9393,B 0,C 0,E1 0.1598,E2 90.071} C_DIS
LIN {X 1.5344,Y -4.4972,Z 16,A -2.9078,B 0,C 0,E1 0.1598,E2 90.0716} C_DIS
LIN {X 2.1724,Y -4.2247,Z 16,A -2.8728,B 0,C 0,E1 0.1598,E2 90.0717} C_DIS
LIN {X 2.8338,Y -3.8112,Z 16,A -2.831,B 0,C 0,E1 0.1598,E2 90.0717} C_DIS
LIN {X 3.4191,Y -3.2959,Z 16,A -2.7876,B 0,C 0,E1 0.1598,E2 90.0717} C_DIS
LIN {X 3.9629,Y -2.6214,Z 16,A -2.7388,B 0,C 0,E1 0.1598,E2 90.0717} C_DIS
LIN {X 4.3015,Y -2.0159,Z 16,A -2.7007,B 0,C 0,E1 0.1598,E2 90.0717} C_DIS
LIN {X 4.5487,Y -1.3679,Z 16,A -2.6641,B 0,C 0,E1 0.1598,E2 90.0717} C_DIS
LIN {X 4.6997,Y -0.691,Z 16,A -2.6298,B 0,C 0,E1 0.1598,E2 90.0718} C_DIS
LIN {X 4.7509,Y 0.0006,Z 16,A -2.5986,B 0,C 0,E1 0.1598,E2 90.0718} C_DIS
LIN {X 4.6999,Y 0.6922,Z 16,A -2.5711,B 0,C 0,E1 0.1598,E2 90.0718} C_DIS
LIN {X 4.5479,Y 1.3689,Z 16,A -2.548,B 0,C 0,E1 0.1598,E2 90.0719} C_DIS
LIN {X 4.3022,Y 2.0174,Z 16,A -2.5296,B 0,C 0,E1 0.1598,E2 90.0719} C_DIS
LIN {X 3.9619,Y 2.6219,Z 16,A -2.5165,B 0,C 0,E1 0.1598,E2 90.072} C_DIS
LIN {X 3.5386,Y 3.1712,Z 16,A -2.5089,B 0,C 0,E1 0.1598,E2 90.072} C_DIS
LIN {X 3.039,Y 3.6525,Z 16,A -2.5069,B 0,C 0,E1 0.1598,E2 90.072} C_DIS
LIN {X 2.4741,Y 4.0547,Z 16,A -2.5107,B 0,C 0,E1 0.1598,E2 90.0721} C_DIS
LIN {X 1.8577,Y 4.3729,Z 16,A -2.52,B 0,C 0,E1 0.1598,E2 90.0721} C_DIS
LIN {X 1.2007,Y 4.5954,Z 16,A -2.5349,B 0,C 0,E1 0.1598,E2 90.0721} C_DIS
LIN {X 0.4325,Y 4.7298,Z 16,A -2.5575,B 0,C 0,E1 0.1598,E2 90.0721} C_DIS
LIN {X -0.5202,Y 4.7227,Z 16,A -2.593,B 0,C 0,E1 0.1598,E2 90.0721} C_DIS
LIN {X -1.2022,Y 4.5964,Z 16,A -2.6234,B 0,C 0,E1 0.1598,E2 90.0721} C_DIS
LIN {X -1.8587,Y 4.3725,Z 16,A -2.6571,B 0,C 0,E1 0.1598,E2 90.0721} C_DIS
LIN {X -2.621,Y 3.9604,Z 16,A -2.7025,B 0,C 0,E1 0.1598,E2 90.0719} C_DIS
LIN {X -3.1695,Y 3.5367,Z 16,A -2.7406,B 0,C 0,E1 0.1598,E2 90.0719} C_DIS
LIN {X -3.6507,Y 3.0376,Z 16,A -2.7794,B 0,C 0,E1 0.1598,E2 90.0717} C_DIS
LIN {X -4.0543,Y 2.4738,Z 16,A -2.818,B 0,C 0,E1 0.1598,E2 90.0717} C_DIS
LIN {X -4.3714,Y 1.857,Z 16,A -2.8556,B 0,C 0,E1 0.1598,E2 90.0716} C_DIS
LIN {X -4.5504,Y 1.3684,Z 16,A -2.8829,B 0,C 0,E1 0.1598,E2 90.0716} C_DIS
LIN {X -4.6999,Y 0.6909,Z 16,A -2.9169,B 0,C 0,E1 0.1598,E2 90.0715} C_DIS
LIN {X -4.75,Y -0.0006,Z 16,A -2.9479,B 0,C 0,E1 0.1598,E2 90.0715} C_DIS
LIN {X -4.6999,Y -0.6921,Z 16,A -2.9752,B 0,C 0,E1 0.1598,E2 90.0714} C_DIS
LIN {X -4.5503,Y -1.3694,Z 16,A -2.9983,B 0,C 0,E1 0.1598,E2 90.0714} C_DIS
LIN {X -4.3031,Y -2.0177,Z 16,A -3.0166,B 0,C 0,E1 0.1598,E2 90.0714} C_DIS
LIN {X -3.9619,Y -2.6217,Z 16,A -3.0296,B 0,C 0,E1 0.1598,E2 90.0714} C_DIS
LIN {X -3.5388,Y -3.1711,Z 16,A -3.0373,B 0,C 0,E1 0.1598,E2 90.0714} C_DIS
LIN {X -3.0393,Y -3.6525,Z 16,A -3.0394,B 0,C 0,E1 0.1598,E2 90.0714} C_DIS
LIN {X -2.4742,Y -4.0545,Z 16,A -3.0357,B 0,C 0,E1 0.1598,E2 90.0714} C_DIS
LIN {X -1.8579,Y -4.3728,Z 16,A -3.0265,B 0,C 0,E1 0.1598,E2 90.0714} C_DIS
LIN {X -1.2009,Y -4.5951,Z 16,A -3.0118,B 0,C 0,E1 0.1598,E2 90.0715} C_DIS
LIN {X -0.5192,Y -4.7222,Z 16,A -2.9922,B 0,C 0,E1 0.1598,E2 90.0715} C_DIS
LIN {X -0.5192,Y -4.7222,Z 16,A -2.9922,B 0,C 0,E1 0.1598,E2 90.0715} C_DIS
Enddeposition()
LIN {X -0.0092,Y -5.6859,Z 16,A -3.0133,B 0,C 0,E1 0.1598,E2 90.0704} C_DIS
Startdeposition()
$VEL.CP = VEL_PRINT
LIN {X -0.7903,Y -5.6306,Z 16,A -3.0407,B 0,C 0,E1 0.1598,E2 90.0715} C_DIS
LIN {X -1.4056,Y -5.5109,Z 16,A -3.0583,B 0,C 0,E1 0.1598,E2 90.0715} C_DIS
LIN {X -2.0033,Y -5.3221,Z 16,A -3.0722,B 0,C 0,E1 0.1598,E2 90.0715} C_DIS
LIN {X -2.7169,Y -4.9987,Z 16,A -3.0847,B 0,C 0,E1 0.1598,E2 90.0714} C_DIS
LIN {X -3.6273,Y -4.3785,Z 16,A -3.0917,B 0,C 0,E1 0.1598,E2 90.0712} C_DIS
Enddeposition()
END
